  MoveL 1037 to (5.94, 339.15, -10) mm, rotated rx 180 ry 0 rz 0.01 deg; joints [44.933, -47.873, 107.559, -131.107, 69.642, 159.025]
  MoveL 1038 to (6.8, 338.95, -10) mm, rotated rx 180 ry 0 rz 0.01 deg; joints [44.952, -47.906, 107.627, -131.098, 69.673, 159.047]
  MoveL 1039 to (7.07, 338.84, -10) mm, rotated rx 180 ry 0 rz 0.01 deg; joints [44.956, -47.917, 107.651, -131.098, 69.683, 159.056]
  MoveL 1040 to (7.57, 338.46, -9.83) mm, rotated rx -180 ry 0 rz 0.01 deg; joints [44.959, -47.953, 107.708, -131.101, 69.698, 159.072]
  MoveL 1041 to (7.78, 338.05, -9.37) mm, rotated rx -180 ry 0 rz 0.01 deg; joints [44.953, -47.996, 107.749, -131.105, 69.694, 159.072]
  MoveL 1042 to (7.82, 337.88, -8.73) mm, rotated rx 180 ry 0 rz 0.01 deg; joints [44.95, -48.036, 107.764, -131.102, 69.677, 159.053]
  Set speed (500.0 mm/s)
  MoveL 1043 to (7.82, 337.88, 11) mm, rotated rx 180 ry 0 rz 0.01 deg; joints [44.942, -49.073, 107.797, -130.824, 69.015, 158.246]
  Set speed (500.0 mm/s)
  MoveL 1044 to (10.27, 334.35, 11) mm, rotated rx -180 ry 0 rz 0.01 deg; joints [44.912, -49.257, 108.178, -130.911, 69.133, 158.417]
  Set speed (100.0 mm/s)
  MoveL 1045 to (10.27, 334.35, -10) mm, rotated rx 180 ry 0 rz 0.01 deg; joints [44.92, -48.148, 108.142, -131.206, 69.84, 159.277]
  MoveL 1046 to (10.27, 31.58, -10) mm, rotated rx 180 ry 0 rz 0.01 deg; joints [35.104, -55.706, 124.759, -143.156, 73.602, 169.001]
  MoveL 1047 to (8.89, 37.17, -10) mm, rotated rx 180 ry 0 rz 0.01 deg; joints [35.276, -55.549, 124.407, -142.947, 73.483, 168.827]
  MoveL 1048 to (8.76, 37.6, -10) mm, rotated rx 180 ry 0 rz 0.01 deg; joints [35.288, -55.536, 124.378, -142.931, 73.473, 168.813]
  MoveL 1049 to (8.49, 38.29, -10) mm, rotated rx 180 ry 0 rz 0.01 deg; joints [35.306, -55.514, 124.328, -142.908, 73.455, 168.79]
  MoveL 1050 to (8.23, 38.81, -10) mm, rotated rx -180 ry 0 rz 0.01 deg; joints [35.319, -55.495, 124.286, -142.891, 73.439, 168.772]
  MoveL 1051 to (2.04, 48.95, -10) mm, rotated rx 180 ry 0 rz 0.01 deg; joints [35.53, -55.095, 123.399, -142.587, 73.098, 168.4]
  MoveL 1052 to (1.89, 49.17, -10) mm, rotated rx 180 ry 0 rz 0.01 deg; joints [35.534, -55.085, 123.378, -142.581, 73.091, 168.392]
  MoveL 1053 to (1.05, 50.33, -10) mm, rotated rx -180 ry 0 rz 0.01 deg; joints [35.555, -55.035, 123.268, -142.549, 73.047, 168.347]
  MoveL 1054 to (0.43, 50.98, -10) mm, rotated rx 180 ry 0 rz 0.01 deg; joints [35.562, -55.003, 123.196, -142.534, 73.018, 168.32]
  MoveL 1055 to (-7.44, 57.3, -10) mm, rotated rx -180 ry 0 rz 0.01 deg; joints [35.587, -54.626, 122.372, -142.424, 72.668, 168.027]
  MoveL 1056 to (-7.81, 57.56, -10) mm, rotated rx 180 ry 0 rz 0.01 deg; joints [35.587, -54.609, 122.335, -142.421, 72.652, 168.014]
  MoveL 1057 to (-8.49, 57.96, -10) mm, rotated rx -180 ry 0 rz 0.01 deg; joints [35.584, -54.58, 122.271, -142.417, 72.624, 167.993]
  MoveL 1058 to (-9.25, 58.3, -10) mm, rotated rx 180 ry 0 rz 0.01 deg; joints [35.577, -54.549, 122.203, -142.418, 72.594, 167.972]
  MoveL 1059 to (-19.1, 61.27, -10) mm, rotated rx -180 ry 0 rz 0.01 deg; joints [35.43, -54.179, 121.402, -142.484, 72.218, 167.743]
  MoveL 1060 to (-19.95, 61.41, -10) mm, rotated rx -180 ry 0 rz 0.01 deg; joints [35.414, -54.15, 121.339, -142.494, 72.187, 167.726]
  MoveL 1061 to (-21.76, 61.48, -10) mm, rotated rx -180 ry 0 rz 0.01 deg; joints [35.37, -54.091, 121.213, -142.526, 72.123, 167.698]
  MoveL 1062 to (-22.2, 61.47, -10) mm, rotated rx -180 ry 0 rz 0.01 deg; joints [35.358, -54.078, 121.185, -142.534, 72.108, 167.691]
  MoveL 1063 to (-29.46, 60.8, -10) mm, rotated rx -180 ry 0 rz 0.01 deg; joints [35.15, -53.864, 120.726, -142.699, 71.865, 167.604]
  MoveL 1064 to (-29.69, 60.77, -10) mm, rotated rx 180 ry 0 rz 0.01 deg; joints [35.144, -53.857, 120.712, -142.704, 71.857, 167.601]
  MoveL 1065 to (-31.5, 60.48, -10) mm, rotated rx 180 ry 0 rz 0.01 deg; joints [35.087, -53.806, 120.603, -142.75, 71.798, 167.583]
  MoveL 1066 to (-32.21, 60.29, -10) mm, rotated rx 180 ry 0 rz 0.01 deg; joints [35.063, -53.788, 120.565, -142.771, 71.776, 167.578]
  MoveL 1067 to (-34.02, 59.57, -10) mm, rotated rx 180 ry 0 rz 0.01 deg; joints [34.991, -53.745, 120.476, -142.835, 71.722, 167.572]
  MoveL 1068 to (-34.31, 59.44, -10) mm, rotated rx 180 ry 0 rz 0.01 deg; joints [34.979, -53.739, 120.462, -142.846, 71.713, 167.571]
  MoveL 1069 to (-41.06, 55.99, -10) mm, rotated rx -180 ry 0 rz 0.01 deg; joints [34.688, -53.597, 120.166, -143.113, 71.52, 167.57]
  MoveL 1070 to (-41.31, 55.85, -10) mm, rotated rx -180 ry 0 rz 0.01 deg; joints [34.676, -53.592, 120.155, -143.124, 71.513, 167.571]
  MoveL 1071 to (-42.24, 55.27, -10) mm, rotated rx 180 ry 0 rz 0.01 deg; joints [34.632, -53.574, 120.119, -143.165, 71.487, 167.574]
  MoveL 1072 to (-42.6, 55.01, -10) mm, rotated rx 180 ry 0 rz 0.01 deg; joints [34.614, -53.568, 120.106, -143.182, 71.478, 167.576]
  MoveL 1073 to (-43.63, 54.17, -10) mm, rotated rx 180 ry 0 rz 0.01 deg; joints [34.559, -53.553, 120.076, -143.236, 71.452, 167.585]
  MoveL 1074 to (-44.02, 53.79, -10) mm, rotated rx 180 ry 0 rz 0.01 deg; joints [34.535, -53.549, 120.067, -143.259, 71.443, 167.59]
  MoveL 1075 to (-46.92, 50.49, -10) mm, rotated rx -180 ry 0 rz 0.01 deg; joints [34.345, -53.525, 120.023, -143.45, 71.382, 167.641]
  MoveL 1076 to (-46.98, 50.42, -10) mm, rotated rx -180 ry 0 rz 0.01 deg; joints [34.341, -53.524, 120.022, -143.454, 71.381, 167.642]
  MoveL 1077 to (-50.32, 46.42, -10) mm, rotated rx -180 ry 0 rz 0.01 deg; joints [34.116, -53.501, 119.98, -143.682, 71.312, 167.707]
  MoveL 1078 to (-50.64, 45.95, -10) mm, rotated rx -180 ry 0 rz 0.01 deg; joints [34.09, -53.5, 119.979, -143.707, 71.306, 167.716]
  MoveL 1079 to (-68.58, 14.91, -10) mm, rotated rx -180 ry 0 rz 0.01 deg; joints [32.531, -53.548, 120.149, -145.334, 71.045, 168.324]
  MoveL 1080 to (-68.71, 14.67, -10) mm, rotated rx 180 ry 0 rz 0.01 deg; joints [32.519, -53.548, 120.15, -145.347, 71.043, 168.329]
  MoveL 1081 to (-69.4, 13.22, -10) mm, rotated rx 180 ry 0 rz 0.01 deg; joints [32.45, -53.555, 120.167, -145.42, 71.036, 168.36]
  MoveL 1082 to (-69.53, 12.89, -10) mm, rotated rx 180 ry 0 rz 0.01 deg; joints [32.434, -53.557, 120.172, -145.437, 71.035, 168.367]
  MoveL 1083 to (-72.09, 5.64, -10) mm, rotated rx 180 ry 0 rz 0.01 deg; joints [32.107, -53.615, 120.314, -145.79, 71.031, 168.529]
  MoveL 1084 to (-72.16, 5.41, -10) mm, rotated rx -180 ry 0 rz 0.01 deg; joints [32.097, -53.618, 120.319, -145.801, 71.031, 168.535]
  MoveL 1085 to (-72.56, 3.96, -10) mm, rotated rx -180 ry 0 rz 0.01 deg; joints [32.034, -53.633, 120.355, -145.87, 71.034, 168.569]
  MoveL 1086 to (-72.66, 3.43, -10) mm, rotated rx 180 ry 0 rz 0.01 deg; joints [32.012, -53.64, 120.371, -145.894, 71.037, 168.582]
  MoveL 1087 to (-72.82, 1.98, -10) mm, rotated rx -180 ry 0 rz 0.01 deg; joints [31.955, -53.663, 120.423, -145.959, 71.048, 168.619]
  MoveL 1088 to (-72.83, 1.45, -10) mm, rotated rx -180 ry 0 rz 0.01 deg; joints [31.935, -53.672, 120.446, -145.982, 71.054, 168.633]
  MoveL 1089 to (-72.48, -5.8, -10) mm, rotated rx 180 ry 0 rz 0.01 deg; joints [31.673, -53.824, 120.786, -146.288, 71.154, 168.835]
  MoveL 1090 to (-72.47, -5.98, -10) mm, rotated rx 180 ry 0 rz 0.01 deg; joints [31.667, -53.828, 120.795, -146.296, 71.157, 168.84]
  MoveL 1091 to (-72.25, -8.15, -10) mm, rotated rx -180 ry 0 rz 0.01 deg; joints [31.59, -53.876, 120.904, -146.386, 71.191, 168.902]
  MoveL 1092 to (-72.12, -8.81, -10) mm, rotated rx -180 ry 0 rz 0.01 deg; joints [31.569, -53.893, 120.942, -146.412, 71.204, 168.921]
  MoveL 1093 to (-71.7, -10.2, -10) mm, rotated rx 180 ry 0 rz 0.01 deg; joints [31.527, -53.934, 121.032, -146.465, 71.236, 168.965]
  MoveL 1094 to (-71.56, -10.56, -10) mm, rotated rx -180 ry 0 rz 0.01 deg; joints [31.516, -53.945, 121.057, -146.478, 71.245, 168.976]
  MoveL 1095 to (-70.7, -12.52, -10) mm, rotated rx -180 ry 0 rz 0.01 deg; joints [31.462, -54.01, 121.202, -146.549, 71.3, 169.041]
  MoveL 1096 to (-70.68, -12.58, -10) mm, rotated rx 180 ry 0 rz 0.01 deg; joints [31.461, -54.012, 121.207, -146.551, 71.301, 169.043]
  MoveL 1097 to (-68.54, -17.21, -10) mm, rotated rx 180 ry 0 rz 0.01 deg; joints [31.335, -54.17, 121.556, -146.716, 71.435, 169.197]
  MoveL 1098 to (-68.48, -17.34, -10) mm, rotated rx -180 ry 0 rz 0.01 deg; joints [31.332, -54.174, 121.565, -146.72, 71.438, 169.201]
  MoveL 1099 to (-67.74, -18.79, -10) mm, rotated rx 180 ry 0 rz 0.01 deg; joints [31.294, -54.226, 121.68, -146.77, 71.483, 169.25]
  MoveL 1100 to (-67.5, -19.18, -10) mm, rotated rx -180 ry 0 rz 0.01 deg; joints [31.285, -54.241, 121.713, -146.783, 71.496, 169.264]
  MoveL 1101 to (-66.73, -20.29, -10) mm, rotated rx -180 ry 0 rz 0.01 deg; joints [31.26, -54.287, 121.814, -146.819, 71.538, 169.304]
  MoveL 1102 to (-66.27, -20.82, -10) mm, rotated rx 180 ry 0 rz 0.01 deg; joints [31.251, -54.312, 121.869, -146.834, 71.561, 169.325]
  MoveL 1103 to (-59.77, -26.97, -10) mm, rotated rx 180 ry 0 rz 0.01 deg; joints [31.167, -54.638, 122.587, -146.991, 71.871, 169.577]
  MoveL 1104 to (-59.61, -27.11, -10) mm, rotated rx 180 ry 0 rz 0.01 deg; joints [31.165, -54.646, 122.603, -146.994, 71.878, 169.583]
  MoveL 1105 to (-58.52, -28.01, -10) mm, rotated rx 180 ry 0 rz 0.01 deg; joints [31.156, -54.698, 122.718, -147.015, 71.928, 169.622]
  MoveC 1106 to (-58.09, -28.32, -10) mm, rotated rx 180 ry 0 rz 0.01 deg; joints [31.154, -54.718, 122.761, -147.021, 71.948, 169.636] to (-57.61, -28.56, -10) mm, rotated rx 180 ry 0 rz 0.01 deg; joints [31.156, -54.738, 122.805, -147.023, 71.968, 169.649]
  MoveL 1107 to (-50.81, -31.27, -10) mm, rotated rx 180 ry 0 rz 0.01 deg; joints [31.21, -55.008, 123.394, -147.024, 72.247, 169.814]
  MoveL 1108 to (-342.73, -31.27, -10) mm, rotated rx -180 ry 0 rz 0.01 deg; joints [25.542, -44.352, 100.839, -150.359, 60.721, 165.533]
  MoveL 1109 to (-336.29, -28.75, -10) mm, rotated rx 180 ry 0 rz 0.01 deg; joints [25.731, -44.57, 101.289, -150.215, 60.975, 165.561]
  MoveL 1110 to (-335.78, -28.5, -10) mm, rotated rx 180 ry 0 rz 0.01 deg; joints [25.748, -44.586, 101.323, -150.201, 60.994, 165.562]
  MoveL 1111 to (-335.05, -28.07, -10) mm, rotated rx -180 ry 0 rz 0.01 deg; joints [25.774, -44.608, 101.367, -150.178, 61.021, 165.56]
  MoveL 1112 to (-334.49, -27.65, -10) mm, rotated rx -180 ry 0 rz 0.01 deg; joints [25.798, -44.623, 101.398, -150.157, 61.041, 165.556]
  MoveL 1113 to (-332.31, -25.62, -10) mm, rotated rx 180 ry 0 rz 0.01 deg; joints [25.902, -44.674, 101.5, -150.057, 61.114, 165.529]
  MoveL 1114 to (-332.27, -25.59, -10) mm, rotated rx -180 ry 0 rz 0.01 deg; joints [25.904, -44.675, 101.502, -150.055, 61.115, 165.529]
  MoveL 1115 to (-326.92, -20.45, -10) mm, rotated rx 180 ry 0 rz 0.01 deg; joints [26.166, -44.796, 101.745, -149.801, 61.293, 165.457]
  MoveL 1116 to (-326.37, -19.77, -10) mm, rotated rx 180 ry 0 rz 0.01 deg; joints [26.198, -44.805, 101.764, -149.768, 61.309, 165.445]
  MoveL 1117 to (-325.69, -18.65, -10) mm, rotated rx 180 ry 0 rz 0.01 deg; joints [26.247, -44.812, 101.775, -149.716, 61.327, 165.421]
  MoveL 1118 to (-325.51, -18.31, -10) mm, rotated rx 180 ry 0 rz 0.01 deg; joints [26.262, -44.813, 101.776, -149.7, 61.331, 165.414]
  MoveL 1119 to (-322.24, -11.28, -10) mm, rotated rx 180 ry 0 rz 0.01 deg; joints [26.553, -44.81, 101.758, -149.376, 61.398, 165.248]
  MoveL 1120 to (-322.12, -11.01, -10) mm, rotated rx -180 ry 0 rz 0.01 deg; joints [26.565, -44.81, 101.756, -149.363, 61.4, 165.241]
  MoveL 1121 to (-321.52, -9.33, -10) mm, rotated rx -180 ry 0 rz 0.01 deg; joints [26.631, -44.802, 101.736, -149.287, 61.408, 165.199]
  MoveL 1122 to (-321.34, -8.57, -10) mm, rotated rx -180 ry 0 rz 0.01 deg; joints [26.66, -44.794, 101.719, -149.253, 61.408, 165.178]
  MoveL 1123 to (-321.05, -6.03, -10) mm, rotated rx -180 ry 0 rz 0.01 deg; joints [26.75, -44.757, 101.635, -149.142, 61.394, 165.103]
  MoveL 1124 to (-321.03, -5.8, -10) mm, rotated rx -180 ry 0 rz 0.01 deg; joints [26.758, -44.753, 101.627, -149.132, 61.392, 165.096]
  MoveL 1125 to (-320.68, 1.45, -10) mm, rotated rx 180 ry 0 rz 0.01 deg; joints [27.007, -44.624, 101.345, -148.816, 61.331, 164.873]
  MoveL 1126 to (-320.69, 1.86, -10) mm, rotated rx -180 ry 0 rz 0.01 deg; joints [27.021, -44.616, 101.327, -148.799, 61.327, 164.86]
  MoveL 1127 to (-320.74, 2.59, -10) mm, rotated rx -180 ry 0 rz 0.01 deg; joints [27.044, -44.599, 101.291, -148.768, 61.317, 164.836]
  MoveL 1128 to (-320.78, 2.94, -10) mm, rotated rx -180 ry 0 rz 0.01 deg; joints [27.055, -44.59, 101.272, -148.753, 61.311, 164.824]
  MoveL 1129 to (-321.05, 4.39, -10) mm, rotated rx 180 ry 0 rz 0.01 deg; joints [27.099, -44.551, 101.187, -148.692, 61.285, 164.773]
  MoveL 1130 to (-321.17, 4.88, -10) mm, rotated rx -180 ry 0 rz 0.01 deg; joints [27.113, -44.536, 101.155, -148.671, 61.274, 164.756]
  MoveL 1131 to (-321.92, 7.06, -10) mm, rotated rx 180 ry 0 rz 0.01 deg; joints [27.173, -44.462, 100.997, -148.582, 61.219, 164.674]
  MoveL 1132 to (-321.94, 7.11, -10) mm, rotated rx 180 ry 0 rz 0.01 deg; joints [27.175, -44.46, 100.993, -148.58, 61.218, 164.672]
  MoveL 1133 to (-324.29, 13.64, -10) mm, rotated rx 180 ry 0 rz 0.01 deg; joints [27.351, -44.233, 100.506, -148.312, 61.048, 164.422]
  MoveL 1134 to (-324.54, 14.18, -10) mm, rotated rx -180 ry 0 rz 0.01 deg; joints [27.365, -44.212, 100.461, -148.29, 61.032, 164.4]
  MoveL 1135 to (-342.52, 45.38, -10) mm, rotated rx -180 ry 0 rz 0.01 deg; joints [28.076, -42.818, 97.505, -147.038, 59.927, 163.048]
  MoveL 1136 to (-342.66, 45.6, -10) mm, rotated rx 180 ry 0 rz 0.01 deg; joints [28.081, -42.808, 97.483, -147.029, 59.919, 163.038]
  MoveL 1137 to (-343.43, 46.73, -10) mm, rotated rx 180 ry 0 rz 0.01 deg; joints [28.104, -42.751, 97.363, -146.983, 59.873, 162.985]
  MoveL 1138 to (-343.65, 47.02, -10) mm, rotated rx -180 ry 0 rz 0.01 deg; joints [28.11, -42.736, 97.33, -146.972, 59.861, 162.971]
  MoveL 1139 to (-348.97, 53.24, -10) mm, rotated rx 180 ry 0 rz 0.01 deg; joints [28.218, -42.378, 96.576, -146.726, 59.563, 162.659]
  MoveL 1140 to (-349.18, 53.47, -10) mm, rotated rx 180 ry 0 rz 0.01 deg; joints [28.222, -42.364, 96.547, -146.718, 59.552, 162.647]
  MoveL 1141 to (-350.19, 54.44, -10) mm, rotated rx 180 ry 0 rz 0.01 deg; joints [28.236, -42.3, 96.413, -146.68, 59.498, 162.595]
  MoveL 1142 to (-350.57, 54.76, -10) mm, rotated rx -180 ry 0 rz 0.01 deg; joints [28.239, -42.277, 96.365, -146.667, 59.477, 162.576]
  MoveL 1143 to (-351.55, 55.47, -10) mm, rotated rx 180 ry 0 rz 0.01 deg; joints [28.245, -42.22, 96.245, -146.641, 59.427, 162.533]
  MoveL 1144 to (-351.98, 55.73, -10) mm, rotated rx -180 ry 0 rz 0.01 deg; joints [28.246, -42.197, 96.196, -146.631, 59.406, 162.516]
  MoveL 1145 to (-359.19, 59.43, -10) mm, rotated rx -180 ry 0 rz 0.01 deg; joints [28.241, -41.809, 95.384, -146.498, 59.051, 162.248]
  MoveL 1146 to (-359.41, 59.54, -10) mm, rotated rx -180 ry 0 rz 0.01 deg; joints [28.24, -41.797, 95.36, -146.495, 59.04, 162.24]
  MoveL 1147 to (-360.86, 60.15, -10) mm, rotated rx 180 ry 0 rz 0.01 deg; joints [28.235, -41.721, 95.202, -146.473, 58.97, 162.19]
  MoveL 1148 to (-361.5, 60.35, -10) mm, rotated rx -180 ry 0 rz 0.01 deg; joints [28.23, -41.69, 95.136, -146.467, 58.94, 162.17]
  MoveL 1149 to (-362.95, 60.65, -10) mm, rotated rx 180 ry 0 rz 0.01 deg; joints [28.215, -41.621, 94.993, -146.458, 58.873, 162.131]
  MoveL 1150 to (-363.32, 60.71, -10) mm, rotated rx 180 ry 0 rz 0.01 deg; joints [28.211, -41.604, 94.957, -146.457, 58.856, 162.122]
  MoveL 1151 to (-371.3, 61.47, -10) mm, rotated rx -180 ry 0 rz 0.01 deg; joints [28.099, -41.243, 94.209, -146.45, 58.495, 161.936]
  MoveL 1152 to (-371.75, 61.48, -10) mm, rotated rx -180 ry 0 rz 0.01 deg; joints [28.092, -41.224, 94.168, -146.451, 58.476, 161.927]
  MoveL 1153 to (-373.56, 61.41, -10) mm, rotated rx 180 ry 0 rz 0.01 deg; joints [28.059, -41.147, 94.009, -146.459, 58.396, 161.892]
  MoveL 1154 to (-374.4, 61.27, -10) mm, rotated rx -180 ry 0 rz 0.01 deg; joints [28.041, -41.114, 93.94, -146.467, 58.36, 161.88]
  MoveL 1155 to (-383.58, 58.54, -10) mm, rotated rx -180 ry 0 rz 0.01 deg; joints [27.801, -40.774, 93.242, -146.61, 57.981, 161.79]
  MoveL 1156 to (-383.9, 58.43, -10) mm, rotated rx 180 ry 0 rz 0.01 deg; joints [27.793, -40.762, 93.218, -146.616, 57.968, 161.788]
  MoveL 1157 to (-384.9, 58.02, -10) mm, rotated rx 180 ry 0 rz 0.01 deg; joints [27.763, -40.728, 93.147, -146.636, 57.927, 161.782]
  MoveL 1158 to (-385.72, 57.54, -10) mm, rotated rx 180 ry 0 rz 0.01 deg; joints [27.734, -40.702, 93.095, -146.659, 57.896, 161.782]
  MoveL 1159 to (-393.23, 51.6, -10) mm, rotated rx -180 ry 0 rz 0.01 deg; joints [27.424, -40.503, 92.693, -146.935, 57.622, 161.838]
  MoveL 1160 to (-393.47, 51.39, -10) mm, rotated rx 180 ry 0 rz 0.01 deg; joints [27.413, -40.497, 92.681, -146.944, 57.613, 161.841]
  MoveL 1161 to (-394.4, 50.5, -10) mm, rotated rx -180 ry 0 rz 0.01 deg; joints [27.37, -40.475, 92.637, -146.985, 57.581, 161.853]
  MoveL 1162 to (-394.94, 49.84, -10) mm, rotated rx 180 ry 0 rz 0.01 deg; joints [27.34, -40.466, 92.62, -147.015, 57.563, 161.866]
  MoveL 1163 to (-401.25, 39.67, -10) mm, rotated rx 180 ry 0 rz 0.01 deg; joints [26.917, -40.408, 92.518, -147.474, 57.386, 162.097]
  MoveL 1164 to (-401.38, 39.45, -10) mm, rotated rx 180 ry 0 rz 0.01 deg; joints [26.908, -40.408, 92.517, -147.483, 57.382, 162.102]
  MoveL 1165 to (-401.99, 38.27, -10) mm, rotated rx -180 ry 0 rz 0.01 deg; joints [26.861, -40.406, 92.515, -147.536, 57.367, 162.131]
  MoveL 1166 to (-402.27, 37.54, -10) mm, rotated rx 180 ry 0 rz 0.01 deg; joints [26.833, -40.409, 92.523, -147.569, 57.362, 162.151]
  MoveL 1167 to (-403.78, 31.65, -10) mm, rotated rx 180 ry 0 rz 0.01 deg; joints [26.622, -40.469, 92.658, -147.831, 57.356, 162.328]
  MoveL 1168 to (-403.79, 333.8, -10) mm, rotated rx 180 ry 0 rz 0.01 deg; joints [35.399, -32.082, 74.938, -134.135, 53.84, 149.634]
  MoveL 1169 to (-403.73, 334.87, -10) mm, rotated rx -180 ry 0 rz 0.01 deg; joints [35.429, -32.047, 74.865, -134.084, 53.829, 149.582]
  MoveL 1170 to (-403.53, 335.74, -10) mm, rotated rx -180 ry 0 rz 0.01 deg; joints [35.455, -32.027, 74.822, -134.044, 53.827, 149.545]
  MoveL 1171 to (-403.42, 336, -10) mm, rotated rx -180 ry 0 rz 0.01 deg; joints [35.464, -32.023, 74.814, -134.032, 53.829, 149.535]
  MoveL 1172 to (-403.03, 336.5, -9.83) mm, rotated rx -180 ry 0 rz 0.01 deg; joints [35.485, -32.032, 74.818, -134.008, 53.836, 149.518]
  MoveL 1173 to (-402.62, 336.71, -9.37) mm, rotated rx -180 ry 0 rz 0.01 deg; joints [35.498, -32.064, 74.846, -133.992, 53.84, 149.506]
  MoveL 1174 to (-402.46, 336.75, -8.73) mm, rotated rx -180 ry 0 rz 0.01 deg; joints [35.502, -32.098, 74.862, -133.979, 53.83, 149.488]
  Set speed (500.0 mm/s)
  MoveL 1175 to (-402.46, 336.75, 11) mm, rotated rx 180 ry 0 rz 0.01 deg; joints [35.493, -32.912, 74.899, -133.574, 53.288, 148.796]
  Set speed (500.0 mm/s)
  MoveL 1176 to (-182.2, 109.36, 11) mm, rotated rx 180 ry 0 rz 0.01 deg; joints [33.246, -48.741, 107.487, -142.719, 64.876, 163.062]
  Set speed (500.0 mm/s)
  MoveL 1177 to (-182.2, 109.36, 1.77) mm, rotated rx 180 ry 0 rz 0.01 deg; joints [33.251, -48.259, 107.475, -142.846, 65.252, 163.373]
  Set speed (100.0 mm/s)
  MoveL 1178 to (-182.04, 109.34, 1.15) mm, rotated rx 180 ry 0 rz 0.01 deg; joints [33.254, -48.233, 107.487, -142.853, 65.284, 163.397]
  MoveL 1179 to (-181.59, 109.31, 0.68) mm, rotated rx -180 ry 0 rz 0.01 deg; joints [33.263, -48.226, 107.521, -142.855, 65.32, 163.421]
  MoveL 1180 to (-180.98, 109.33, 0.5) mm, rotated rx -180 ry 0 rz 0.01 deg; joints [33.277, -48.238, 107.567, -142.85, 65.35, 163.437]
  MoveL 1181 to (-175.74, 113.35, 0.26) mm, rotated rx -180 ry 0 rz 0.01 deg; joints [33.523, -48.323, 107.762, -142.624, 65.514, 163.401]
  MoveL 1182 to (-177.33, 119.76, 0.01) mm, rotated rx 180 ry 0 rz 0.01 deg; joints [33.698, -48.103, 107.32, -142.379, 65.392, 163.174]
  MoveL 1183 to (-183.84, 120.88, -0.23) mm, rotated rx -180 ry 0 rz 0.01 deg; joints [33.593, -47.827, 106.771, -142.412, 65.143, 163.038]
  MoveL 1184 to (-187.47, 115.36, -0.48) mm, rotated rx -180 ry 0 rz 0.01 deg; joints [33.336, -47.81, 106.772, -142.686, 65.077, 163.166]
  MoveL 1185 to (-183.86, 109.82, -0.72) mm, rotated rx -180 ry 0 rz 0.01 deg; joints [33.232, -48.057, 107.321, -142.879, 65.285, 163.414]
  MoveL 1186 to (-177.35, 110.91, -0.96) mm, rotated rx -180 ry 0 rz 0.01 deg; joints [33.408, -48.257, 107.76, -142.761, 65.53, 163.494]
  MoveL 1187 to (-175.73, 117.31, -1.21) mm, rotated rx -180 ry 0 rz 0.01 deg; joints [33.653, -48.154, 107.562, -142.479, 65.529, 163.322]
  MoveL 1188 to (-180.95, 121.36, -1.45) mm, rotated rx -180 ry 0 rz 0.01 deg; joints [33.672, -47.857, 106.963, -142.375, 65.296, 163.111]
  MoveL 1189 to (-186.75, 118.2, -1.7) mm, rotated rx -180 ry 0 rz 0.01 deg; joints [33.444, -47.706, 106.682, -142.576, 65.121, 163.126]
  MoveL 1190 to (-186.18, 111.62, -1.94) mm, rotated rx -180 ry 0 rz 0.01 deg; joints [33.242, -47.867, 107.053, -142.847, 65.226, 163.358]
  MoveL 1191 to (-179.92, 109.5, -2.18) mm, rotated rx 180 ry 0 rz 0.01 deg; joints [33.307, -48.131, 107.633, -142.866, 65.497, 163.538]
  MoveL 1192 to (-175.48, 114.39, -2.43) mm, rotated rx -180 ry 0 rz 0.01 deg; joints [33.564, -48.167, 107.724, -142.613, 65.621, 163.462]
  MoveL 1193 to (-178.17, 120.42, -2.67) mm, rotated rx 180 ry 0 rz 0.01 deg; joints [33.702, -47.916, 107.218, -142.398, 65.461, 163.229]
  MoveL 1194 to (-184.77, 120.37, -2.92) mm, rotated rx 180 ry 0 rz 0.01 deg; joints [33.558, -47.664, 106.72, -142.48, 65.221, 163.129]
  MoveL 1195 to (-187.37, 114.3, -3.16) mm, rotated rx 180 ry 0 rz 0.01 deg; joints [33.304, -47.698, 106.826, -142.766, 65.2, 163.292]
  MoveL 1196 to (-182.85, 109.48, -3.4) mm, rotated rx -180 ry 0 rz 0.01 deg; joints [33.244, -47.961, 107.409, -142.918, 65.436, 163.531]
  MoveL 1197 to (-176.63, 111.69, -3.65) mm, rotated rx -180 ry 0 rz 0.01 deg; joints [33.451, -48.123, 107.769, -142.756, 65.657, 163.57]
  MoveL 1198 to (-176.16, 118.28, -3.89) mm, rotated rx 180 ry 0 rz 0.01 deg; joints [33.677, -47.975, 107.475, -142.479, 65.61, 163.373]
  MoveL 1199 to (-182.01, 121.35, -4.14) mm, rotated rx 180 ry 0 rz 0.01 deg; joints [33.65, -47.678, 106.878, -142.424, 65.363, 163.184]
  MoveL 1200 to (-187.17, 117.22, -4.38) mm, rotated rx -180 ry 0 rz 0.01 deg; joints [33.405, -47.574, 106.693, -142.658, 65.224, 163.24]
  MoveL 1201 to (-185.45, 110.84, -4.63) mm, rotated rx 180 ry 0 rz 0.01 deg; joints [33.234, -47.771, 107.142, -142.907, 65.371, 163.484]
  MoveL 1202 to (-178.92, 109.86, -4.87) mm, rotated rx -180 ry 0 rz 0.01 deg; joints [33.342, -48.018, 107.685, -142.875, 65.64, 163.632]
  MoveL 1203 to (-175.4, 115.45, -5.11) mm, rotated rx 180 ry 0 rz 0.01 deg; joints [33.602, -48.003, 107.671, -142.604, 65.72, 163.518]
  MoveL 1204 to (-179.11, 120.91, -5.36) mm, rotated rx -180 ry 0 rz 0.01 deg; joints [33.699, -47.73, 107.116, -142.424, 65.527, 163.287]
  MoveL 1205 to (-185.61, 119.7, -5.6) mm, rotated rx 180 ry 0 rz 0.01 deg; joints [33.52, -47.509, 106.685, -142.553, 65.304, 163.226]
  MoveL 1206 to (-187.1, 113.27, -5.85) mm, rotated rx -180 ry 0 rz 0.01 deg; joints [33.278, -47.591, 106.893, -142.841, 65.33, 163.419]
  MoveL 1207 to (-181.8, 109.32, -6.09) mm, rotated rx -180 ry 0 rz 0.01 deg; joints [33.263, -47.861, 107.491, -142.948, 65.586, 163.643]
  MoveL 1208 to (-176.06, 112.6, -6.33) mm, rotated rx -180 ry 0 rz 0.01 deg; joints [33.494, -47.981, 107.761, -142.747, 65.777, 163.64]
  MoveL 1209 to (-176.76, 119.16, -6.58) mm, rotated rx -180 ry 0 rz 0.01 deg; joints [33.694, -47.791, 107.379, -142.486, 65.685, 163.424]
  MoveL 1210 to (-183.06, 121.15, -6.82) mm, rotated rx 180 ry 0 rz 0.01 deg; joints [33.623, -47.504, 106.802, -142.48, 65.433, 163.262]
  MoveL 1211 to (-187.41, 116.18, -7.07) mm, rotated rx 180 ry 0 rz 0.01 deg; joints [33.367, -47.448, 106.721, -142.74, 65.333, 163.359]
  MoveL 1212 to (-184.59, 110.21, -7.31) mm, rotated rx -180 ry 0 rz 0.01 deg; joints [33.233, -47.675, 107.232, -142.959, 65.519, 163.608]
  MoveL 1213 to (-177.99, 110.39, -7.55) mm, rotated rx -180 ry 0 rz 0.01 deg; joints [33.381, -47.897, 107.723, -142.877, 65.778, 163.72]
  MoveL 1214 to (-175.52, 116.51, -7.8) mm, rotated rx 180 ry 0 rz 0.01 deg; joints [33.635, -47.833, 107.603, -142.597, 65.812, 163.572]
  MoveL 1215 to (-180.13, 121.24, -8.04) mm, rotated rx -180 ry 0 rz 0.01 deg; joints [33.689, -47.544, 107.017, -142.459, 65.592, 163.349]
  MoveL 1216 to (-186.31, 118.9, -8.29) mm, rotated rx 180 ry 0 rz 0.01 deg; joints [33.48, -47.362, 106.665, -142.631, 65.393, 163.329]
  MoveL 1217 to (-186.64, 112.3, -8.53) mm, rotated rx 180 ry 0 rz 0.01 deg; joints [33.258, -47.489, 106.969, -142.912, 65.466, 163.546]
  MoveL 1218 to (-180.73, 109.35, -8.77) mm, rotated rx 180 ry 0 rz 0.01 deg; joints [33.288, -47.758, 107.564, -142.969, 65.735, 163.748]
  MoveL 1219 to (-175.66, 113.59, -9.02) mm, rotated rx -180 ry 0 rz 0.01 deg; joints [33.537, -47.831, 107.735, -142.736, 65.889, 163.704]
  MoveL 1220 to (-177.51, 119.93, -9.26) mm, rotated rx 180 ry 0 rz 0.01 deg; joints [33.704, -47.605, 107.278, -142.498, 65.755, 163.476]
  MoveL 1221 to (-184.06, 120.78, -9.51) mm, rotated rx -180 ry 0 rz 0.01 deg; joints [33.59, -47.336, 106.738, -142.543, 65.506, 163.347]
  MoveL 1222 to (-187.46, 115.12, -9.75) mm, rotated rx -180 ry 0 rz 0.01 deg; joints [33.333, -47.33, 106.763, -142.82, 65.451, 163.481]
  MoveL 1223 to (-183.64, 109.73, -9.99) mm, rotated rx 180 ry 0 rz 0.01 deg; joints [33.239, -47.579, 107.322, -143.003, 65.669, 163.728]
  MoveL 1224 to (-177.17, 111.07, -10.24) mm, rotated rx 180 ry 0 rz 0.01 deg; joints [33.423, -47.769, 107.743, -142.874, 65.91, 163.8]
  MoveL 1225 to (-175.81, 117.54, -10.48) mm, rotated rx 180 ry 0 rz 0.01 deg; joints [33.664, -47.657, 107.522, -142.593, 65.896, 163.623]
  MoveL 1226 to (-181.19, 121.37, -10.73) mm, rotated rx -180 ry 0 rz 0.01 deg; joints [33.672, -47.362, 106.923, -142.501, 65.657, 163.416]
  MoveL 1227 to (-186.86, 117.98, -10.97) mm, rotated rx 180 ry 0 rz 0.01 deg; joints [33.44, -47.222, 106.662, -142.711, 65.489, 163.438]
  MoveL 1228 to (-186.03, 111.43, -11.21) mm, rotated rx -180 ry 0 rz 0.01 deg; joints [33.244, -47.39, 107.052, -142.976, 65.607, 163.673]
  MoveL 1229 to (-179.69, 109.57, -11.46) mm, rotated rx -180 ry 0 rz 0.01 deg; joints [33.32, -47.648, 107.625, -142.983, 65.88, 163.847]
  MoveL 1230 to (-175.44, 114.63, -11.7) mm, rotated rx 180 ry 0 rz 0.01 deg; joints [33.577, -47.672, 107.693, -142.725, 65.993, 163.763]
  MoveL 1231 to (-178.38, 120.55, -11.95) mm, rotated rx -180 ry 0 rz 0.01 deg; joints [33.707, -47.418, 107.174, -142.518, 65.822, 163.531]
  MoveL 1232 to (-184.97, 120.23, -12.19) mm, rotated rx 180 ry 0 rz 0.01 deg; joints [33.554, -47.174, 106.689, -142.612, 65.584, 163.437]
  MoveL 1233 to (-187.33, 114.06, -12.43) mm, rotated rx -180 ry 0 rz 0.01 deg; joints [33.303, -47.218, 106.819, -142.898, 65.575, 163.606]
  MoveL 1234 to (-182.62, 109.43, -12.68) mm, rotated rx -180 ry 0 rz 0.01 deg; joints [33.253, -47.481, 107.407, -143.039, 65.819, 163.843]
  MoveL 1235 to (-176.49, 111.89, -12.92) mm, rotated rx -180 ry 0 rz 0.01 deg; joints [33.466, -47.633, 107.747, -142.867, 66.034, 163.874]
  MoveL 1236 to (-176.29, 118.49, -13.17) mm, rotated rx 180 ry 0 rz 0.01 deg; joints [33.686, -47.476, 107.431, -142.594, 65.975, 163.673]
  MoveL 1237 to (-182.26, 121.32, -13.41) mm, rotated rx -180 ry 0 rz 0.01 deg; joints [33.649, -47.183, 106.837, -142.551, 65.724, 163.488]
  MoveL 1238 to (-187.24, 116.99, -13.65) mm, rotated rx 180 ry 0 rz 0.01 deg; joints [33.401, -47.09, 106.676, -142.791, 65.593, 163.552]
  MoveL 1239 to (-185.26, 110.68, -13.9) mm, rotated rx -180 ry 0 rz 0.01 deg; joints [33.237, -47.293, 107.14, -143.033, 65.752, 163.798]
  MoveL 1240 to (-178.7, 109.97, -14.14) mm, rotated rx -180 ry 0 rz 0.01 deg; joints [33.355, -47.532, 107.672, -142.989, 66.021, 163.939]
  MoveL 1241 to (-175.41, 115.7, -14.39) mm, rotated rx 180 ry 0 rz 0.01 deg; joints [33.615, -47.506, 107.634, -142.715, 66.089, 163.818]
  MoveL 1242 to (-179.34, 121, -14.63) mm, rotated rx 180 ry 0 rz 0.01 deg; joints [33.702, -47.231, 107.07, -142.546, 65.887, 163.588]
  MoveL 1243 to (-185.78, 119.53, -14.87) mm, rotated rx -180 ry 0 rz 0.01 deg; joints [33.515, -47.02, 106.655, -142.685, 65.668, 163.535]
  MoveL 1244 to (-187.01, 113.04, -15.12) mm, rotated rx 180 ry 0 rz 0.01 deg; joints [33.278, -47.112, 106.886, -142.972, 65.706, 163.732]
  MoveL 1245 to (-181.56, 109.31, -15.36) mm, rotated rx 180 ry 0 rz 0.01 deg; joints [33.273, -47.38, 107.485, -143.066, 65.969, 163.952]
  MoveL 1246 to (-175.96, 112.82, -15.61) mm, rotated rx -180 ry 0 rz 0.01 deg; joints [33.509, -47.488, 107.733, -142.857, 66.151, 163.942]
  MoveL 1247 to (-176.92, 119.35, -15.85) mm, rotated rx -180 ry 0 rz 0.01 deg; joints [33.702, -47.291, 107.332, -142.601, 66.047, 163.723]
  MoveL 1248 to (-183.29, 121.08, -16.1) mm, rotated rx 180 ry 0 rz 0.01 deg; joints [33.62, -47.01, 106.762, -142.608, 65.793, 163.567]
  MoveL 1249 to (-187.44, 115.94, -16.34) mm, rotated rx 180 ry 0 rz 0.01 deg; joints [33.364, -46.965, 106.705, -142.872, 65.704, 163.671]
  MoveL 1250 to (-184.38, 110.08, -16.58) mm, rotated rx 180 ry 0 rz 0.01 deg; joints [33.238, -47.196, 107.228, -143.083, 65.9, 163.919]
  MoveL 1251 to (-177.79, 110.53, -16.83) mm, rotated rx 180 ry 0 rz 0.01 deg; joints [33.395, -47.409, 107.704, -142.989, 66.157, 164.024]
  MoveL 1252 to (-175.57, 116.75, -17.07) mm, rotated rx -180 ry 0 rz 0.01 deg; joints [33.647, -47.334, 107.561, -142.708, 66.178, 163.87]
  MoveL 1253 to (-180.37, 121.28, -17.32) mm, rotated rx 180 ry 0 rz 0.01 deg; joints [33.691, -47.045, 106.97, -142.581, 65.951, 163.65]
  MoveL 1254 to (-186.45, 118.7, -17.56) mm, rotated rx -180 ry 0 rz 0.01 deg; joints [33.476, -46.874, 106.638, -142.762, 65.758, 163.638]
  MoveL 1255 to (-186.52, 112.09, -17.8) mm, rotated rx -180 ry 0 rz 0.01 deg; joints [33.259, -47.009, 106.962, -143.04, 65.843, 163.858]
  MoveL 1256 to (-180.49, 109.39, -18.05) mm, rotated rx 180 ry 0 rz 0.01 deg; joints [33.3, -47.273, 107.553, -143.084, 66.117, 164.055]
  MoveL 1257 to (-175.6, 113.82, -18.29) mm, rotated rx -180 ry 0 rz 0.01 deg; joints [33.551, -47.335, 107.701, -142.845, 66.261, 164.004]
  MoveL 1258 to (-177.7, 120.08, -18.54) mm, rotated rx 180 ry 0 rz 0.01 deg; joints [33.71, -47.104, 107.228, -142.615, 66.116, 163.774]
  MoveL 1259 to (-184.28, 120.67, -18.78) mm, rotated rx 180 ry 0 rz 0.01 deg; joints [33.587, -46.842, 106.7, -142.671, 65.866, 163.651]
  MoveL 1260 to (-187.45, 114.87, -19.02) mm, rotated rx 180 ry 0 rz 0.01 deg; joints [33.33, -46.848, 106.749, -142.951, 65.823, 163.792]
  MoveL 1261 to (-183.41, 109.65, -19.27) mm, rotated rx -180 ry 0 rz 0.01 deg; joints [33.246, -47.098, 107.315, -143.124, 66.05, 164.037]
  MoveL 1262 to (-177, 111.25, -19.51) mm, rotated rx 180 ry 0 rz 0.01 deg; joints [33.437, -47.278, 107.719, -142.984, 66.287, 164.102]
  MoveL 1263 to (-175.91, 117.76, -19.76) mm, rotated rx 180 ry 0 rz 0.01 deg; joints [33.674, -47.156, 107.476, -142.704, 66.26, 163.92]
  MoveL 1264 to (-181.43, 121.38, -20) mm, rotated rx -180 ry 0 rz 0.01 deg; joints [33.672, -46.863, 106.875, -142.624, 66.015, 163.717]
  MoveL 1265 to (-213.98, 121.38, -20) mm, rotated rx 180 ry 0 rz 0.01 deg; joints [32.98, -45.681, 104.376, -142.983, 64.753, 163.15]
  MoveC 1266 to (-215.9, 120.27, -20) mm, rotated rx 180 ry 0 rz 0.01 deg; joints [32.904, -45.636, 104.282, -143.049, 64.69, 163.153] to (-215.9, 118.04, -20) mm, rotated rx -180 ry 0 rz 0.01 deg; joints [32.833, -45.687, 104.394, -143.142, 64.717, 163.226]
  MoveL 1267 to (-214.81, 116.14, -20) mm, rotated rx 180 ry 0 rz 0.01 deg; joints [32.794, -45.771, 104.575, -143.21, 64.782, 163.308]
  MoveC 1268 to (-213.77, 115.1, -20) mm, rotated rx 180 ry 0 rz 0.01 deg; joints [32.782, -45.833, 104.708, -143.242, 64.835, 163.36] to (-212.35, 114.72, -20) mm, rotated rx -180 ry 0 rz 0.01 deg; joints [32.799, -45.894, 104.838, -143.243, 64.895, 163.397]
  MoveL 1269 to (-181.15, 114.72, -20) mm, rotated rx 180 ry 0 rz 0.01 deg; joints [33.461, -47.025, 107.231, -142.896, 66.106, 163.936]
  MoveC 1270 to (-179.73, 115.1, -20) mm, rotated rx 180 ry 0 rz 0.01 deg; joints [33.505, -47.067, 107.319, -142.863, 66.156, 163.948] to (-178.69, 116.14, -20) mm, rotated rx 180 ry 0 rz 0.01 deg; joints [33.561, -47.081, 107.346, -142.808, 66.183, 163.932]
  MoveL 1271 to (-177.6, 118.04, -20) mm, rotated rx 180 ry 0 rz 0.01 deg; joints [33.647, -47.077, 107.334, -142.716, 66.202, 163.89]
  MoveC 1272 to (-177.59, 120.26, -20) mm, rotated rx 180 ry 0 rz 0.01 deg; joints [33.719, -47.026, 107.222, -142.624, 66.176, 163.818] to (-179.52, 121.38, -20) mm, rotated rx 180 ry 0 rz 0.01 deg; joints [33.714, -46.932, 107.02, -142.601, 66.088, 163.749]
  MoveL 1273 to (-181.43, 121.38, -20) mm, rotated rx -180 ry 0 rz 0.01 deg; joints [33.672, -46.863, 106.875, -142.624, 66.015, 163.717]
  MoveC 1274 to (-184.81, 122.4, -20) mm, rotated rx 180 ry 0 rz 0.01 deg; joints [33.632, -46.719, 106.568, -142.621, 65.873, 163.626] to (-187.05, 125.12, -20) mm, rotated rx 180 ry 0 rz 0.01 deg; joints [33.672, -46.576, 106.26, -142.535, 65.755, 163.498]
  MoveC 1275 to (-189.29, 127.84, -20) mm, rotated rx 180 ry 0 rz 0.01 deg; joints [33.712, -46.432, 105.951, -142.448, 65.636, 163.37] to (-192.66, 128.86, -20) mm, rotated rx 180 ry 0 rz 0.01 deg; joints [33.672, -46.286, 105.641, -142.444, 65.494, 163.278]
  MoveL 1276 to (-214.9, 128.86, -20) mm, rotated rx 180 ry 0 rz 0.01 deg; joints [33.201, -45.473, 103.925, -142.682, 64.628, 162.886]
  MoveC 1277 to (-218.57, 128.97, -20) mm, rotated rx -180 ry 0 rz 0.01 deg; joints [33.128, -45.335, 103.633, -142.715, 64.483, 162.816] to (-222.23, 129.28, -20) mm, rotated rx -180 ry 0 rz 0.01 deg; joints [33.062, -45.191, 103.33, -142.738, 64.334, 162.74]
  MoveC 1278 to (-225.89, 129.69, -20) mm, rotated rx 180 ry 0 rz 0.01 deg; joints [32.999, -45.046, 103.022, -142.756, 64.185, 162.66] to (-229.54, 130.08, -20) mm, rotated rx 180 ry 0 rz 0.01 deg; joints [32.936, -44.9, 102.713, -142.775, 64.036, 162.581]
  MoveC 1279 to (-231.34, 129.16, -20) mm, rotated rx -180 ry 0 rz 0.01 deg; joints [32.87, -44.854, 102.618, -142.83, 63.975, 162.579] to (-231.23, 127.15, -20) mm, rotated rx -180 ry 0 rz 0.01 deg; joints [32.808, -44.905, 102.73, -142.913, 64.003, 162.649]
  MoveC 1280 to (-228.5, 123.23, -20) mm, rotated rx 180 ry 0 rz 0.01 deg; joints [32.739, -45.098, 103.144, -143.051, 64.158, 162.829] to (-225.92, 119.22, -20) mm, rotated rx 180 ry 0 rz 0.01 deg; joints [32.663, -45.288, 103.55, -143.193, 64.308, 163.009]
  MoveC 1281 to (-223.44, 115.14, -20) mm, rotated rx 180 ry 0 rz 0.01 deg; joints [32.583, -45.474, 103.95, -143.339, 64.454, 163.188] to (-221.03, 111.02, -20) mm, rotated rx 180 ry 0 rz 0.01 deg; joints [32.5, -45.657, 104.345, -143.486, 64.597, 163.366]
  MoveC 1282 to (-217.92, 107.91, -20) mm, rotated rx 180 ry 0 rz 0.01 deg; joints [32.463, -45.843, 104.742, -143.584, 64.757, 163.522] to (-213.68, 106.78, -20) mm, rotated rx 180 ry 0 rz 0.01 deg; joints [32.514, -46.025, 105.13, -143.588, 64.937, 163.633]
  MoveL 1283 to (-179.83, 106.78, -20) mm, rotated rx -180 ry 0 rz 0.01 deg; joints [33.229, -47.252, 107.726, -143.209, 66.251, 164.213]
  MoveC 1284 to (-175.59, 107.91, -20) mm, rotated rx -180 ry 0 rz 0.01 deg; joints [33.359, -47.377, 107.99, -143.111, 66.4, 164.248] to (-172.47, 111.02, -20) mm, rotated rx 180 ry 0 rz 0.01 deg; joints [33.528, -47.418, 108.07, -142.944, 66.482, 164.202]
  MoveC 1285 to (-170.06, 115.13, -20) mm, rotated rx -180 ry 0 rz 0.01 deg; joints [33.716, -47.41, 108.046, -142.745, 66.524, 164.111] to (-167.6, 119.21, -20) mm, rotated rx -180 ry 0 rz 0.01 deg; joints [33.904, -47.404, 108.026, -142.546, 66.569, 164.022]
  MoveC 1286 to (-165.03, 123.23, -20) mm, rotated rx 180 ry 0 rz 0.01 deg; joints [34.091, -47.403, 108.016, -142.348, 66.618, 163.937] to (-162.31, 127.14, -20) mm, rotated rx 180 ry 0 rz 0.01 deg; joints [34.279, -47.409, 108.021, -142.153, 66.674, 163.857]
  MoveC 1287 to (-162.2, 129.16, -20) mm, rotated rx 180 ry 0 rz 0.01 deg; joints [34.347, -47.366, 107.926, -142.069, 66.654, 163.793] to (-164.01, 130.08, -20) mm, rotated rx 180 ry 0 rz 0.01 deg; joints [34.337, -47.281, 107.745, -142.054, 66.574, 163.733]
  MoveC 1288 to (-167.65, 129.69, -20) mm, rotated rx 180 ry 0 rz 0.01 deg; joints [34.244, -47.161, 107.492, -142.115, 66.441, 163.683] to (-171.3, 129.28, -20) mm, rotated rx 180 ry 0 rz 0.01 deg; joints [34.15, -47.042, 107.24, -142.176, 66.307, 163.634]
  MoveC 1289 to (-174.95, 128.97, -20) mm, rotated rx 180 ry 0 rz 0.01 deg; joints [34.06, -46.919, 106.981, -142.234, 66.172, 163.582] to (-178.62, 128.86, -20) mm, rotated rx -180 ry 0 rz 0.01 deg; joints [33.976, -46.791, 106.709, -142.282, 66.033, 163.522]
  MoveL 1290 to (-192.66, 128.86, -20) mm, rotated rx -180 ry 0 rz 0.01 deg; joints [33.672, -46.286, 105.641, -142.444, 65.494, 163.278]
  MoveC 1291 to (-195.95, 129.86, -20) mm, rotated rx -180 ry 0 rz 0.01 deg; joints [33.634, -46.144, 105.339, -142.439, 65.355, 163.188] to (-198.13, 132.51, -20) mm, rotated rx 180 ry 0 rz 0.01 deg; joints [33.672, -46.003, 105.036, -142.354, 65.239, 163.062]
  MoveC 1292 to (-200.31, 135.16, -20) mm, rotated rx 180 ry 0 rz 0.01 deg; joints [33.711, -45.862, 104.733, -142.268, 65.122, 162.936] to (-203.6, 136.15, -20) mm, rotated rx 180 ry 0 rz 0.01 deg; joints [33.673, -45.718, 104.428, -142.262, 64.983, 162.844]
  MoveL 1293 to (-214.9, 136.15, -20) mm, rotated rx -180 ry 0 rz 0.01 deg; joints [33.434, -45.303, 103.552, -142.379, 64.542, 162.642]
  MoveC 1294 to (-223.13, 136.48, -20) mm, rotated rx 180 ry 0 rz 0.01 deg; joints [33.272, -44.989, 102.89, -142.448, 64.214, 162.482] to (-231.31, 137.45, -20) mm, rotated rx -180 ry 0 rz 0.01 deg; joints [33.133, -44.659, 102.195, -142.485, 63.879, 162.3]
  MoveC 1295 to (-239.44, 138.81, -20) mm, rotated rx -180 ry 0 rz 0.01 deg; joints [33.009, -44.32, 101.479, -142.503, 63.539, 162.103] to (-247.53, 140.32, -20) mm, rotated rx 180 ry 0 rz 0.01 deg; joints [32.891, -43.976, 100.753, -142.51, 63.197, 161.9]
  MoveC 1296 to (-249.26, 139.53, -20) mm, rotated rx 180 ry 0 rz 0.01 deg; joints [32.831, -43.928, 100.655, -142.558, 63.137, 161.894] to (-249.09, 137.64, -20) mm, rotated rx 180 ry 0 rz 0.01 deg; joints [32.776, -43.98, 100.767, -142.635, 63.166, 161.963]
  MoveC 1297 to (-243.73, 131.29, -20) mm, rotated rx 180 ry 0 rz 0.01 deg; joints [32.684, -44.335, 101.524, -142.854, 63.456, 162.28] to (-238.53, 124.81, -20) mm, rotated rx 180 ry 0 rz 0.01 deg; joints [32.584, -44.684, 102.269, -143.079, 63.74, 162.594]
  MoveC 1298 to (-233.64, 118.08, -20) mm, rotated rx -180 ry 0 rz 0.01 deg; joints [32.469, -45.024, 102.998, -143.314, 64.014, 162.908] to (-229.24, 111.03, -20) mm, rotated rx 180 ry 0 rz 0.01 deg; joints [32.332, -45.351, 103.699, -143.567, 64.272, 163.22]
  MoveC 1299 to (-228.22, 109.2, -20) mm, rotated rx -180 ry 0 rz 0.01 deg; joints [32.294, -45.431, 103.87, -143.633, 64.334, 163.299] to (-227.27, 107.34, -20) mm, rotated rx -180 ry 0 rz 0.01 deg; joints [32.253, -45.509, 104.038, -143.702, 64.394, 163.377]
  MoveC 1300 to (-226.31, 105.48, -20) mm, rotated rx 180 ry 0 rz 0.01 deg; joints [32.212, -45.587, 104.206, -143.77, 64.454, 163.455] to (-225.29, 103.65, -20) mm, rotated rx 180 ry 0 rz 0.01 deg; joints [32.174, -45.666, 104.376, -143.836, 64.515, 163.532]
  MoveC 1301 to (-222.18, 100.54, -20) mm, rotated rx -180 ry 0 rz 0.01 deg; joints [32.136, -45.851, 104.773, -143.935, 64.675, 163.688] to (-217.94, 99.4, -20) mm, rotated rx -180 ry 0 rz 0.01 deg; joints [32.186, -46.034, 105.161, -143.94, 64.856, 163.799]
  MoveL 1302 to (-175.58, 99.4, -20) mm, rotated rx 180 ry 0 rz 0.01 deg; joints [33.078, -47.568, 108.41, -143.464, 66.502, 164.518]
  MoveC 1303 to (-171.33, 100.54, -20) mm, rotated rx 180 ry 0 rz 0.01 deg; joints [33.207, -47.693, 108.674, -143.364, 66.651, 164.553] to (-168.22, 103.65, -20) mm, rotated rx -180 ry 0 rz 0.01 deg; joints [33.378, -47.734, 108.755, -143.197, 66.733, 164.507]
  MoveC 1304 to (-167.14, 105.59, -20) mm, rotated rx -180 ry 0 rz 0.01 deg; joints [33.466, -47.728, 108.74, -143.103, 66.75, 164.463] to (-166.12, 107.56, -20) mm, rotated rx -180 ry 0 rz 0.01 deg; joints [33.553, -47.72, 108.719, -143.009, 66.765, 164.418]
  MoveC 1305 to (-165.1, 109.53, -20) mm, rotated rx 180 ry 0 rz 0.01 deg; joints [33.64, -47.712, 108.697, -142.914, 66.78, 164.373] to (-164.02, 111.47, -20) mm, rotated rx -180 ry 0 rz 0.01 deg; joints [33.728, -47.706, 108.681, -142.821, 66.798, 164.329]
  MoveC 1306 to (-159.67, 118.42, -20) mm, rotated rx 180 ry 0 rz 0.01 deg; joints [34.052, -47.701, 108.658, -142.479, 66.879, 164.181] to (-154.84, 125.04, -20) mm, rotated rx 180 ry 0 rz 0.01 deg; joints [34.377, -47.719, 108.683, -142.144, 66.981, 164.05]
  MoveC 1307 to (-149.7, 131.41, -20) mm, rotated rx 180 ry 0 rz 0.01 deg; joints [34.7, -47.751, 108.739, -141.815, 67.097, 163.932] to (-144.39, 137.65, -20) mm, rotated rx 180 ry 0 rz 0.01 deg; joints [35.023, -47.79, 108.81, -141.489, 67.219, 163.821]
  MoveC 1308 to (-144.2, 139.54, -20) mm, rotated rx 180 ry 0 rz 0.01 deg; joints [35.089, -47.752, 108.727, -141.409, 67.203, 163.763] to (-145.93, 140.33, -20) mm, rotated rx -180 ry 0 rz 0.01 deg; joints [35.075, -47.674, 108.559, -141.4, 67.129, 163.708]
  MoveC 1309 to (-154.04, 138.82, -20) mm, rotated rx 180 ry 0 rz 0.01 deg; joints [34.843, -47.427, 108.038, -141.568, 66.844, 163.619] to (-162.17, 137.45, -20) mm, rotated rx 180 ry 0 rz 0.01 deg; joints [34.616, -47.174, 107.504, -141.728, 66.555, 163.525]
  MoveC 1310 to (-170.37, 136.48, -20) mm, rotated rx -180 ry 0 rz 0.01 deg; joints [34.403, -46.907, 106.941, -141.869, 66.256, 163.415] to (-178.62, 136.15, -20) mm, rotated rx -180 ry 0 rz 0.01 deg; joints [34.211, -46.621, 106.337, -141.981, 65.946, 163.283]
  MoveL 1311 to (-203.6, 136.15, -20) mm, rotated rx 180 ry 0 rz 0.01 deg; joints [33.673, -45.718, 104.428, -142.262, 64.983, 162.844]
  MoveC 1312 to (-206.7, 137.09, -20) mm, rotated rx 180 ry 0 rz 0.01 deg; joints [33.637, -45.583, 104.141, -142.256, 64.851, 162.758] to (-208.75, 139.59, -20) mm, rotated rx 180 ry 0 rz 0.01 deg; joints [33.673, -45.448, 103.853, -142.174, 64.741, 162.637]
  MoveC 1313 to (-210.81, 142.09, -20) mm, rotated rx -180 ry 0 rz 0.01 deg; joints [33.708, -45.313, 103.564, -142.092, 64.631, 162.516] to (-213.9, 143.02, -20) mm, rotated rx 180 ry 0 rz 0.01 deg; joints [33.673, -45.177, 103.274, -142.085, 64.499, 162.429]
  MoveL 1314 to (-214.9, 143.02, -20) mm, rotated rx -180 ry 0 rz 0.01 deg; joints [33.652, -45.14, 103.197, -142.095, 64.46, 162.411]
  MoveC 1315 to (-230.2, 143.85, -20) mm, rotated rx 180 ry 0 rz 0.01 deg; joints [33.358, -44.549, 101.951, -142.208, 63.847, 162.102] to (-245.33, 146.33, -20) mm, rotated rx 180 ry 0 rz 0.01 deg; joints [33.125, -43.916, 100.617, -142.24, 63.215, 161.734]
  MoveC 1316 to (-260.13, 150.28, -20) mm, rotated rx -180 ry 0 rz 0.01 deg; joints [32.948, -43.251, 99.214, -142.196, 62.572, 161.314] to (-274.52, 155.53, -20) mm, rotated rx -180 ry 0 rz 0.01 deg; joints [32.822, -42.559, 97.756, -142.081, 61.923, 160.845]
  MoveC 1317 to (-276.08, 155, -20) mm, rotated rx 180 ry 0 rz 0.01 deg; joints [32.775, -42.511, 97.655, -142.114, 61.866, 160.833] to (-275.75, 153.39, -20) mm, rotated rx 180 ry 0 rz 0.01 deg; joints [32.732, -42.563, 97.768, -142.18, 61.898, 160.897]
  MoveC 1318 to (-266.78, 146.05, -20) mm, rotated rx 180 ry 0 rz 0.01 deg; joints [32.683, -43.094, 98.893, -142.424, 62.351, 161.333] to (-258.39, 138.07, -20) mm, rotated rx -180 ry 0 rz 0.01 deg; joints [32.602, -43.612, 99.993, -142.694, 62.786, 161.772]
  MoveC 1319 to (-250.57, 129.52, -20) mm, rotated rx -180 ry 0 rz 0.01 deg; joints [32.49, -44.116, 101.066, -142.988, 63.202, 162.213] to (-243.33, 120.47, -20) mm, rotated rx 180 ry 0 rz 0.01 deg; joints [32.348, -44.603, 102.106, -143.303, 63.599, 162.653]
  MoveC 1320 to (-241.11, 117.37, -20) mm, rotated rx 180 ry 0 rz 0.01 deg; joints [32.294, -44.759, 102.44, -143.413, 63.724, 162.797] to (-239.02, 114.19, -20) mm, rotated rx 180 ry 0 rz 0.01 deg; joints [32.235, -44.911, 102.766, -143.527, 63.845, 162.941]
  MoveC 1321 to (-237.02, 110.95, -20) mm, rotated rx 180 ry 0 rz 0.01 deg; joints [32.171, -45.061, 103.087, -143.644, 63.963, 163.084] to (-235.09, 107.67, -20) mm, rotated rx -180 ry 0 rz 0.01 deg; joints [32.104, -45.208, 103.404, -143.763, 64.079, 163.227]
  MoveC 1322 to (-233.59, 104.97, -20) mm, rotated rx -180 ry 0 rz 0.01 deg; joints [32.048, -45.326, 103.657, -143.862, 64.17, 163.343] to (-232.17, 102.22, -20) mm, rotated rx -180 ry 0 rz 0.01 deg; joints [31.987, -45.441, 103.904, -143.963, 64.259, 163.458]
  MoveC 1323 to (-230.76, 99.48, -20) mm, rotated rx 180 ry 0 rz 0.01 deg; joints [31.927, -45.555, 104.151, -144.064, 64.347, 163.572] to (-229.26, 96.78, -20) mm, rotated rx -180 ry 0 rz 0.01 deg; joints [31.87, -45.672, 104.402, -144.163, 64.438, 163.687]
  MoveC 1324 to (-226.15, 93.67, -20) mm, rotated rx 180 ry 0 rz 0.01 deg; joints [31.831, -45.857, 104.798, -144.262, 64.598, 163.841] to (-221.91, 92.53, -20) mm, rotated rx 180 ry 0 rz 0.01 deg; joints [31.88, -46.04, 105.186, -144.267, 64.78, 163.951]
  MoveL 1325 to (-171.61, 92.53, -20) mm, rotated rx 180 ry 0 rz 0.01 deg; joints [32.935, -47.86, 109.044, -143.7, 66.736, 164.8]
  MoveC 1326 to (-167.36, 93.67, -20) mm, rotated rx 180 ry 0 rz 0.01 deg; joints [33.065, -47.985, 109.308, -143.6, 66.885, 164.834] to (-164.25, 96.78, -20) mm, rotated rx 180 ry 0 rz 0.01 deg; joints [33.236, -48.026, 109.388, -143.432, 66.966, 164.788]
  MoveC 1327 to (-162.69, 99.58, -20) mm, rotated rx -180 ry 0 rz 0.01 deg; joints [33.364, -48.019, 109.368, -143.295, 66.992, 164.726] to (-161.22, 102.44, -20) mm, rotated rx -180 ry 0 rz 0.01 deg; joints [33.491, -48.007, 109.338, -143.158, 67.013, 164.661]
  MoveC 1328 to (-159.74, 105.29, -20) mm, rotated rx -180 ry 0 rz 0.01 deg; joints [33.618, -47.995, 109.307, -143.022, 67.035, 164.596] to (-158.18, 108.09, -20) mm, rotated rx 180 ry 0 rz 0.01 deg; joints [33.745, -47.987, 109.284, -142.885, 67.06, 164.533]
  MoveC 1329 to (-149.84, 120.91, -20) mm, rotated rx -180 ry 0 rz 0.01 deg; joints [34.354, -47.987, 109.261, -142.248, 67.219, 164.266] to (-140.18, 132.76, -20) mm, rotated rx 180 ry 0 rz 0.01 deg; joints [34.96, -48.048, 109.369, -141.633, 67.435, 164.049]
  MoveC 1330 to (-129.41, 143.6, -20) mm, rotated rx -180 ry 0 rz 0.01 deg; joints [35.561, -48.164, 109.596, -141.041, 67.702, 163.881] to (-117.71, 153.43, -20) mm, rotated rx 180 ry 0 rz 0.01 deg; joints [36.153, -48.329, 109.929, -140.475, 68.01, 163.759]
  MoveC 1331 to (-117.39, 155.04, -20) mm, rotated rx -180 ry 0 rz 0.01 deg; joints [36.212, -48.302, 109.867, -140.405, 68.002, 163.712] to (-118.95, 155.56, -20) mm, rotated rx -180 ry 0 rz 0.01 deg; joints [36.192, -48.237, 109.728, -140.407, 67.939, 163.669]
  MoveC 1332 to (-129.3, 151.62, -20) mm, rotated rx 180 ry 0 rz 0.01 deg; joints [35.823, -47.979, 109.187, -140.713, 67.608, 163.623] to (-139.9, 148.43, -20) mm, rotated rx 180 ry 0 rz 0.01 deg; joints [35.475, -47.691, 108.581, -140.989, 67.255, 163.547]
  MoveC 1333 to (-150.7, 145.97, -20) mm, rotated rx -180 ry 0 rz 0.01 deg; joints [35.149, -47.375, 107.916, -141.232, 66.883, 163.443] to (-161.62, 144.16, -20) mm, rotated rx 180 ry 0 rz 0.01 deg; joints [34.845, -47.036, 107.199, -141.446, 66.494, 163.315]
  MoveC 1334 to (-170.1, 143.31, -20) mm, rotated rx -180 ry 0 rz 0.01 deg; joints [34.629, -46.756, 106.609, -141.585, 66.184, 163.196] to (-178.62, 143.02, -20) mm, rotated rx 180 ry 0 rz 0.01 deg; joints [34.432, -46.46, 105.983, -141.699, 65.863, 163.057]
  MoveL 1335 to (-213.9, 143.02, -20) mm, rotated rx -180 ry 0 rz 0.01 deg; joints [33.673, -45.177, 103.274, -142.085, 64.499, 162.429]
  MoveC 1336 to (-216.88, 143.93, -20) mm, rotated rx -180 ry 0 rz 0.01 deg; joints [33.639, -45.045, 102.995, -142.077, 64.372, 162.344] to (-218.85, 146.35, -20) mm, rotated rx -180 ry 0 rz 0.01 deg; joints [33.674, -44.914, 102.715, -141.996, 64.266, 162.226]
  MoveC 1337 to (-220.76, 148.78, -20) mm, rotated rx -180 ry 0 rz 0.01 deg; joints [33.71, -44.784, 102.438, -141.914, 64.162, 162.108] to (-223.68, 149.82, -20) mm, rotated rx 180 ry 0 rz 0.01 deg; joints [33.682, -44.65, 102.154, -141.899, 64.034, 162.019]
  MoveC 1338 to (-236.97, 151.3, -20) mm, rotated rx 180 ry 0 rz 0.01 deg; joints [33.452, -44.114, 101.024, -141.96, 63.49, 161.72] to (-250.06, 154.05, -20) mm, rotated rx 180 ry 0 rz 0.01 deg; joints [33.269, -43.548, 99.83, -141.958, 62.934, 161.376]
  MoveC 1339 to (-266.96, 159.49, -20) mm, rotated rx -180 ry 0 rz 0.01 deg; joints [33.095, -42.758, 98.166, -141.861, 62.186, 160.854] to (-283.14, 166.82, -20) mm, rotated rx -180 ry 0 rz 0.01 deg; joints [32.997, -41.937, 96.435, -141.663, 61.436, 160.266]
  MoveC 1340 to (-285.4, 166.75, -20) mm, rotated rx -180 ry 0 rz 0.01 deg; joints [32.95, -41.848, 96.25, -141.68, 61.344, 160.222] to (-286.51, 164.78, -20) mm, rotated rx -180 ry 0 rz 0.01 deg; joints [32.869, -41.853, 96.264, -141.77, 61.321, 160.271]
  MoveL 1341 to (-286.5, 156.62, -20) mm, rotated rx -180 ry 0 rz 0.01 deg; joints [32.619, -42.056, 96.702, -142.115, 61.417, 160.566]
  MoveC 1342 to (-285.74, 153.49, -20) mm, rotated rx -180 ry 0 rz 0.01 deg; joints [32.538, -42.164, 96.933, -142.242, 61.485, 160.693] to (-283.63, 151.06, -20) mm, rotated rx 180 ry 0 rz 0.01 deg; joints [32.505, -42.308, 97.238, -142.331, 61.601, 160.823]
  MoveC 1343 to (-271.09, 141.19, -20) mm, rotated rx -180 ry 0 rz 0.01 deg; joints [32.446, -43.043, 98.794, -142.66, 62.232, 161.419] to (-259.61, 130.1, -20) mm, rotated rx -180 ry 0 rz 0.01 deg; joints [32.327, -43.754, 100.305, -143.038, 62.83, 162.024]
  MoveC 1344 to (-249.39, 117.83, -20) mm, rotated rx -180 ry 0 rz 0.01 deg; joints [32.142, -44.434, 101.755, -143.467, 63.386, 162.631] to (-240.63, 104.47, -20) mm, rotated rx 180 ry 0 rz 0.01 deg; joints [31.889, -45.072, 103.122, -143.949, 63.894, 163.234]
  MoveC 1345 to (-238.68, 100.95, -20) mm, rotated rx -180 ry 0 rz 0.01 deg; joints [31.815, -45.225, 103.452, -144.078, 64.014, 163.385] to (-236.83, 97.36, -20) mm, rotated rx -180 ry 0 rz 0.01 deg; joints [31.736, -45.375, 103.774, -144.211, 64.129, 163.535]
  MoveC 1346 to (-234.98, 93.78, -20) mm, rotated rx 180 ry 0 rz 0.01 deg; joints [31.656, -45.524, 104.096, -144.344, 64.245, 163.684] to (-233.03, 90.26, -20) mm, rotated rx -180 ry 0 rz 0.01 deg; joints [31.581, -45.676, 104.422, -144.473, 64.364, 163.832]
  MoveC 1347 to (-229.92, 87.15, -20) mm, rotated rx -180 ry 0 rz 0.01 deg; joints [31.541, -45.861, 104.818, -144.573, 64.524, 163.986] to (-225.68, 86.01, -20) mm, rotated rx -180 ry 0 rz 0.01 deg; joints [31.59, -46.044, 105.207, -144.578, 64.706, 164.096]
  MoveL 1348 to (-167.85, 86.01, -20) mm, rotated rx 180 ry 0 rz 0.01 deg; joints [32.798, -48.135, 109.642, -143.924, 66.958, 165.064]
  MoveC 1349 to (-163.6, 87.15, -20) mm, rotated rx 180 ry 0 rz 0.01 deg; joints [32.929, -48.26, 109.905, -143.823, 67.106, 165.099] to (-160.49, 90.26, -20) mm, rotated rx -180 ry 0 rz 0.01 deg; joints [33.101, -48.301, 109.987, -143.654, 67.187, 165.053]
  MoveC 1350 to (-158.47, 93.89, -20) mm, rotated rx 180 ry 0 rz 0.01 deg; joints [33.266, -48.292, 109.961, -143.477, 67.22, 164.974] to (-156.56, 97.57, -20) mm, rotated rx 180 ry 0 rz 0.01 deg; joints [33.432, -48.277, 109.922, -143.3, 67.248, 164.89]
  MoveC 1351 to (-154.66, 101.26, -20) mm, rotated rx 180 ry 0 rz 0.01 deg; joints [33.597, -48.262, 109.883, -143.122, 67.275, 164.806] to (-152.63, 104.89, -20) mm, rotated rx 180 ry 0 rz 0.01 deg; joints [33.762, -48.252, 109.854, -142.945, 67.308, 164.726]
  MoveC 1352 to (-143.93, 118.14, -20) mm, rotated rx 180 ry 0 rz 0.01 deg; joints [34.395, -48.255, 109.835, -142.283, 67.474, 164.452] to (-133.78, 130.31, -20) mm, rotated rx 180 ry 0 rz 0.01 deg; joints [35.026, -48.325, 109.962, -141.645, 67.703, 164.234]
  MoveC 1353 to (-122.37, 141.3, -20) mm, rotated rx 180 ry 0 rz 0.01 deg; joints [35.65, -48.458, 110.224, -141.035, 67.989, 164.073] to (-109.9, 151.07, -20) mm, rotated rx -180 ry 0 rz 0.01 deg; joints [36.261, -48.648, 110.611, -140.456, 68.324, 163.966]
  MoveC 1354 to (-107.77, 153.5, -20) mm, rotated rx 180 ry 0 rz 0.01 deg; joints [36.391, -48.661, 110.635, -140.326, 68.371, 163.923] to (-107.01, 156.64, -20) mm, rotated rx -180 ry 0 rz 0.01 deg; joints [36.51, -48.612, 110.525, -140.188, 68.36, 163.834]
  MoveL 1355 to (-107.01, 164.77, -20) mm, rotated rx -180 ry 0 rz 0.01 deg; joints [36.772, -48.417, 110.095, -139.86, 68.259, 163.57]
  MoveC 1356 to (-108.12, 166.73, -20) mm, rotated rx -180 ry 0 rz 0.01 deg; joints [36.808, -48.333, 109.912, -139.797, 68.195, 163.487] to (-110.37, 166.8, -20) mm, rotated rx -180 ry 0 rz 0.01 deg; joints [36.756, -48.256, 109.748, -139.828, 68.112, 163.447]
  MoveC 1357 to (-122.79, 160.99, -20) mm, rotated rx 180 ry 0 rz 0.01 deg; joints [36.276, -47.976, 109.165, -140.242, 67.731, 163.427] to (-135.72, 156.41, -20) mm, rotated rx -180 ry 0 rz 0.01 deg; joints [35.828, -47.645, 108.469, -140.607, 67.312, 163.357]
  MoveC 1358 to (-148.99, 152.98, -20) mm, rotated rx 180 ry 0 rz 0.01 deg; joints [35.413, -47.268, 107.676, -140.924, 66.861, 163.242] to (-162.49, 150.62, -20) mm, rotated rx 180 ry 0 rz 0.01 deg; joints [35.033, -46.852, 106.798, -141.192, 66.383, 163.087]
  MoveC 1359 to (-170.54, 149.81, -20) mm, rotated rx -180 ry 0 rz 0.01 deg; joints [34.827, -46.587, 106.239, -141.324, 66.089, 162.974] to (-178.62, 149.54, -20) mm, rotated rx -180 ry 0 rz 0.01 deg; joints [34.64, -46.305, 105.644, -141.431, 65.785, 162.841]
  MoveL 1360 to (-214.9, 149.54, -20) mm, rotated rx -180 ry 0 rz 0.01 deg; joints [33.858, -44.984, 102.857, -141.825, 64.383, 162.19]
  MoveC 1361 to (-219.29, 149.61, -20) mm, rotated rx 180 ry 0 rz 0.01 deg; joints [33.767, -44.819, 102.51, -141.865, 64.21, 162.107] to (-223.68, 149.82, -20) mm, rotated rx 180 ry 0 rz 0.01 deg; joints [33.682, -44.65, 102.154, -141.899, 64.034, 162.019]
  MoveC 1362 to (-227.3, 151.19, -20) mm, rotated rx 180 ry 0 rz 0.01 deg; joints [33.649, -44.482, 101.797, -141.877, 63.875, 161.905] to (-229.54, 154.35, -20) mm, rotated rx 180 ry 0 rz 0.01 deg; joints [33.701, -44.321, 101.454, -141.766, 63.749, 161.754]
  MoveC 1363 to (-231.69, 157.53, -20) mm, rotated rx -180 ry 0 rz 0.01 deg; joints [33.756, -44.162, 101.115, -141.654, 63.626, 161.604] to (-235.2, 159.11, -20) mm, rotated rx 180 ry 0 rz 0.01 deg; joints [33.732, -43.991, 100.753, -141.62, 63.468, 161.483]
  MoveC 1364 to (-257.17, 164.18, -20) mm, rotated rx 180 ry 0 rz 0.01 deg; joints [33.437, -43.024, 98.715, -141.591, 62.528, 160.881] to (-278.03, 172.73, -20) mm, rotated rx 180 ry 0 rz 0.01 deg; joints [33.279, -41.991, 96.539, -141.381, 61.577, 160.155]
  MoveC 1365 to (-281.48, 174.62, -20) mm, rotated rx 180 ry 0 rz 0.01 deg; joints [33.267, -41.806, 96.149, -141.324, 61.413, 160.016] to (-284.78, 176.74, -20) mm, rotated rx -180 ry 0 rz 0.01 deg; joints [33.266, -41.62, 95.757, -141.255, 61.251, 159.869]
  MoveC 1366 to (-288.03, 178.95, -20) mm, rotated rx 180 ry 0 rz 0.01 deg; joints [33.268, -41.433, 95.364, -141.181, 61.091, 159.72] to (-291.31, 181.11, -20) mm, rotated rx -180 ry 0 rz 0.01 deg; joints [33.269, -41.246, 94.969, -141.109, 60.929, 159.571]
  MoveC 1367 to (-293.48, 181.19, -20) mm, rotated rx 180 ry 0 rz 0.01 deg; joints [33.228, -41.156, 94.781, -141.117, 60.838, 159.522] to (-294.59, 179.32, -20) mm, rotated rx 180 ry 0 rz 0.01 deg; joints [33.15, -41.159, 94.79, -141.203, 60.814, 159.568]
  MoveL 1368 to (-294.58, 153.81, -20) mm, rotated rx -180 ry 0 rz 0.01 deg; joints [32.375, -41.802, 96.175, -142.283, 61.115, 160.502]
  MoveC 1369 to (-293.49, 149.38, -20) mm, rotated rx -180 ry 0 rz 0.01 deg; joints [32.261, -41.955, 96.502, -142.464, 61.212, 160.684] to (-290.45, 145.97, -20) mm, rotated rx -180 ry 0 rz 0.01 deg; joints [32.215, -42.16, 96.937, -142.59, 61.378, 160.868]
  MoveC 1370 to (-280.55, 138.56, -20) mm, rotated rx -180 ry 0 rz 0.01 deg; joints [32.178, -42.734, 98.151, -142.838, 61.874, 161.327] to (-271.33, 130.31, -20) mm, rotated rx -180 ry 0 rz 0.01 deg; joints [32.101, -43.293, 99.338, -143.119, 62.35, 161.794]
  MoveC 1371 to (-262.81, 121.34, -20) mm, rotated rx -180 ry 0 rz 0.01 deg; joints [31.987, -43.836, 100.492, -143.431, 62.802, 162.263] to (-255.03, 111.73, -20) mm, rotated rx 180 ry 0 rz 0.01 deg; joints [31.835, -44.358, 101.607, -143.771, 63.23, 162.732]
  MoveC 1372 to (-251.15, 106.2, -20) mm, rotated rx -180 ry 0 rz 0.01 deg; joints [31.735, -44.633, 102.195, -143.97, 63.451, 162.988] to (-247.6, 100.45, -20) mm, rotated rx 180 ry 0 rz 0.01 deg; joints [31.621, -44.898, 102.764, -144.18, 63.661, 163.242]
  MoveC 1373 to (-245.07, 95.92, -20) mm, rotated rx 180 ry 0 rz 0.01 deg; joints [31.524, -45.096, 103.189, -144.348, 63.816, 163.436] to (-242.65, 91.32, -20) mm, rotated rx -180 ry 0 rz 0.01 deg; joints [31.423, -45.29, 103.607, -144.519, 63.966, 163.629]
  MoveC 1374 to (-240.23, 86.71, -20) mm, rotated rx -180 ry 0 rz 0.01 deg; joints [31.321, -45.483, 104.022, -144.69, 64.117, 163.821] to (-237.7, 82.18, -20) mm, rotated rx -180 ry 0 rz 0.01 deg; joints [31.223, -45.678, 104.443, -144.856, 64.271, 164.012]
  MoveC 1375 to (-234.59, 79.07, -20) mm, rotated rx -180 ry 0 rz 0.01 deg; joints [31.182, -45.863, 104.838, -144.957, 64.432, 164.165] to (-230.35, 77.93, -20) mm, rotated rx -180 ry 0 rz 0.01 deg; joints [31.23, -46.046, 105.227, -144.964, 64.615, 164.274]
  MoveL 1376 to (-163.19, 77.93, -20) mm, rotated rx 180 ry 0 rz 0.01 deg; joints [32.627, -48.474, 110.379, -144.202, 67.232, 165.389]
  MoveC 1377 to (-158.94, 79.07, -20) mm, rotated rx 180 ry 0 rz 0.01 deg; joints [32.758, -48.598, 110.641, -144.099, 67.38, 165.423] to (-155.83, 82.18, -20) mm, rotated rx 180 ry 0 rz 0.01 deg; joints [32.931, -48.639, 110.723, -143.929, 67.461, 165.378]
  MoveC 1378 to (-153.23, 86.82, -20) mm, rotated rx -180 ry 0 rz 0.01 deg; joints [33.144, -48.629, 110.693, -143.702, 67.504, 165.278] to (-150.74, 91.52, -20) mm, rotated rx 180 ry 0 rz 0.01 deg; joints [33.357, -48.613, 110.649, -143.474, 67.541, 165.173]
  MoveC 1379 to (-148.26, 96.22, -20) mm, rotated rx 180 ry 0 rz 0.01 deg; joints [33.57, -48.596, 110.603, -143.246, 67.577, 165.068] to (-145.66, 100.86, -20) mm, rotated rx 180 ry 0 rz 0.01 deg; joints [33.783, -48.583, 110.567, -143.019, 67.619, 164.966]
  MoveC 1380 to (-137.06, 113.9, -20) mm, rotated rx -180 ry 0 rz 0.01 deg; joints [34.411, -48.587, 110.551, -142.364, 67.782, 164.699] to (-126.97, 125.83, -20) mm, rotated rx -180 ry 0 rz 0.01 deg; joints [35.036, -48.66, 110.684, -141.733, 68.009, 164.489]
  MoveC 1381 to (-115.6, 136.53, -20) mm, rotated rx 180 ry 0 rz 0.01 deg; joints [35.653, -48.798, 110.957, -141.131, 68.295, 164.337] to (-103.12, 145.92, -20) mm, rotated rx -180 ry 0 rz 0.01 deg; joints [36.255, -48.996, 111.362, -140.563, 68.633, 164.244]
  MoveC 1382 to (-100.04, 149.33, -20) mm, rotated rx 180 ry 0 rz 0.01 deg; joints [36.44, -49.018, 111.403, -140.378, 68.702, 164.186] to (-98.93, 153.79, -20) mm, rotated rx 180 ry 0 rz 0.01 deg; joints [36.612, -48.949, 111.248, -140.181, 68.687, 164.061]
  MoveL 1383 to (-98.93, 179.33, -20) mm, rotated rx -180 ry 0 rz 0.01 deg; joints [37.432, -48.332, 109.888, -139.153, 68.37, 163.228]
  MoveC 1384 to (-100.03, 181.19, -20) mm, rotated rx 180 ry 0 rz 0.01 deg; joints [37.464, -48.25, 109.709, -139.095, 68.307, 163.148] to (-102.2, 181.11, -20) mm, rotated rx 180 ry 0 rz 0.01 deg; joints [37.409, -48.18, 109.56, -139.131, 68.23, 163.114]
  MoveC 1385 to (-109.98, 176.31, -20) mm, rotated rx 180 ry 0 rz 0.01 deg; joints [37.069, -48.037, 109.266, -139.439, 68.009, 163.14] to (-117.96, 171.85, -20) mm, rotated rx 180 ry 0 rz 0.01 deg; joints [36.737, -47.877, 108.935, -139.734, 67.774, 163.152]
  MoveC 1386 to (-126.22, 167.91, -20) mm, rotated rx -180 ry 0 rz 0.01 deg; joints [36.416, -47.693, 108.55, -140.01, 67.521, 163.141] to (-134.79, 164.69, -20) mm, rotated rx 180 ry 0 rz 0.01 deg; joints [36.114, -47.477, 108.099, -140.258, 67.245, 163.1]
  MoveC 1387 to (-154.43, 159.86, -20) mm, rotated rx -180 ry 0 rz 0.01 deg; joints [35.509, -46.914, 106.912, -140.713, 66.574, 162.921] to (-174.56, 157.99, -20) mm, rotated rx -180 ry 0 rz 0.01 deg; joints [34.998, -46.247, 105.507, -141.037, 65.837, 162.63]
  MoveL 1388 to (-214.9, 157.62, -20) mm, rotated rx 180 ry 0 rz 0.01 deg; joints [34.111, -44.789, 102.432, -141.49, 64.287, 161.914]
  MoveC 1389 to (-225.08, 158, -20) mm, rotated rx 180 ry 0 rz 0.01 deg; joints [33.908, -44.4, 101.614, -141.573, 63.882, 161.712] to (-235.2, 159.11, -20) mm, rotated rx -180 ry 0 rz 0.01 deg; joints [33.732, -43.991, 100.753, -141.62, 63.468, 161.483]
  MoveC 1390 to (-238.61, 160.73, -20) mm, rotated rx 180 ry 0 rz 0.01 deg; joints [33.711, -43.822, 100.395, -141.582, 63.313, 161.361] to (-240.52, 163.99, -20) mm, rotated rx 180 ry 0 rz 0.01 deg; joints [33.773, -43.669, 100.069, -141.464, 63.199, 161.211]
  MoveC 1391 to (-242.34, 167.26, -20) mm, rotated rx 180 ry 0 rz 0.01 deg; joints [33.836, -43.519, 99.747, -141.343, 63.087, 161.06] to (-245.61, 169.1, -20) mm, rotated rx 180 ry 0 rz 0.01 deg; joints [33.825, -43.348, 99.386, -141.294, 62.934, 160.932]
  MoveC 1392 to (-260.38, 173.55, -20) mm, rotated rx 180 ry 0 rz 0.01 deg; joints [33.659, -42.665, 97.948, -141.224, 62.287, 160.482] to (-274.53, 179.7, -20) mm, rotated rx 180 ry 0 rz 0.01 deg; joints [33.56, -41.953, 96.449, -141.065, 61.638, 159.973]
  MoveC 1393 to (-281.08, 183.31, -20) mm, rotated rx 180 ry 0 rz 0.01 deg; joints [33.538, -41.6, 95.705, -140.955, 61.326, 159.704] to (-287.33, 187.43, -20) mm, rotated rx 180 ry 0 rz 0.01 deg; joints [33.537, -41.243, 94.953, -140.819, 61.019, 159.421]
  MoveC 1394 to (-293.36, 191.85, -20) mm, rotated rx -180 ry 0 rz 0.01 deg; joints [33.55, -40.884, 94.197, -140.666, 60.717, 159.126] to (-299.27, 196.42, -20) mm, rotated rx 180 ry 0 rz 0.01 deg; joints [33.569, -40.523, 93.437, -140.502, 60.416, 158.825]
  MoveC 1395 to (-301.34, 196.65, -20) mm, rotated rx 180 ry 0 rz 0.01 deg; joints [33.536, -40.433, 93.248, -140.502, 60.327, 158.771] to (-302.44, 194.89, -20) mm, rotated rx 180 ry 0 rz 0.01 deg; joints [33.462, -40.434, 93.253, -140.582, 60.302, 158.814]
  MoveL 1396 to (-302.44, 149.18, -20) mm, rotated rx -180 ry 0 rz 0.01 deg; joints [32.082, -41.598, 95.757, -142.524, 60.84, 160.509]
  MoveC 1397 to (-301.34, 144.93, -20) mm, rotated rx -180 ry 0 rz 0.01 deg; joints [31.972, -41.747, 96.075, -142.699, 60.936, 160.684] to (-298.33, 141.75, -20) mm, rotated rx -180 ry 0 rz 0.01 deg; joints [31.932, -41.946, 96.498, -142.816, 61.099, 160.86]
  MoveC 1398 to (-287.88, 134.43, -20) mm, rotated rx 180 ry 0 rz 0.01 deg; joints [31.907, -42.542, 97.756, -143.061, 61.62, 161.328] to (-278.22, 126.09, -20) mm, rotated rx 180 ry 0 rz 0.01 deg; joints [31.834, -43.123, 98.987, -143.347, 62.116, 161.807]
  MoveC 1399 to (-269.37, 116.91, -20) mm, rotated rx 180 ry 0 rz 0.01 deg; joints [31.717, -43.684, 100.181, -143.669, 62.586, 162.291] to (-261.31, 107.02, -20) mm, rotated rx -180 ry 0 rz 0.01 deg; joints [31.561, -44.224, 101.333, -144.021, 63.029, 162.775]
  MoveC 1400 to (-257.7, 101.88, -20) mm, rotated rx 180 ry 0 rz 0.01 deg; joints [31.467, -44.48, 101.881, -144.207, 63.236, 163.012] to (-254.41, 96.53, -20) mm, rotated rx 180 ry 0 rz 0.01 deg; joints [31.359, -44.727, 102.41, -144.404, 63.431, 163.249]
  MoveC 1401 to (-251.3, 91.01, -20) mm, rotated rx 180 ry 0 rz 0.01 deg; joints [31.242, -44.969, 102.929, -144.609, 63.621, 163.486] to (-248.32, 85.43, -20) mm, rotated rx -180 ry 0 rz 0.01 deg; joints [31.119, -45.206, 103.439, -144.818, 63.806, 163.721]
  MoveC 1402 to (-245.34, 79.84, -20) mm, rotated rx -180 ry 0 rz 0.01 deg; joints [30.995, -45.441, 103.946, -145.026, 63.991, 163.954] to (-242.23, 74.32, -20) mm, rotated rx -180 ry 0 rz 0.01 deg; joints [30.875, -45.678, 104.457, -145.229, 64.18, 164.185]
  MoveC 1403 to (-239.13, 71.22, -20) mm, rotated rx -180 ry 0 rz 0.01 deg; joints [30.833, -45.862, 104.852, -145.331, 64.341, 164.338] to (-234.89, 70.08, -20) mm, rotated rx 180 ry 0 rz 0.01 deg; joints [30.88, -46.046, 105.242, -145.338, 64.524, 164.446]
  MoveL 1404 to (-158.66, 70.08, -20) mm, rotated rx -180 ry 0 rz 0.01 deg; joints [32.459, -48.8, 111.089, -144.471, 67.499, 165.702]
  MoveC 1405 to (-154.41, 71.22, -20) mm, rotated rx 180 ry 0 rz 0.01 deg; joints [32.59, -48.924, 111.351, -144.367, 67.647, 165.735] to (-151.3, 74.33, -20) mm, rotated rx -180 ry 0 rz 0.01 deg; joints [32.764, -48.966, 111.434, -144.196, 67.727, 165.69]
  MoveL 1406 to (-138.86, 96.93, -20) mm, rotated rx 180 ry 0 rz 0.01 deg; joints [33.804, -48.904, 111.259, -143.089, 67.921, 165.199]
  MoveC 1407 to (-130.1, 110.06, -20) mm, rotated rx 180 ry 0 rz 0.01 deg; joints [34.442, -48.911, 111.249, -142.424, 68.087, 164.933] to (-119.73, 121.97, -20) mm, rotated rx -180 ry 0 rz 0.01 deg; joints [35.077, -48.994, 111.402, -141.786, 68.323, 164.73]
  MoveC 1408 to (-108.01, 132.54, -20) mm, rotated rx -180 ry 0 rz 0.01 deg; joints [35.7, -49.145, 111.704, -141.181, 68.621, 164.589] to (-95.19, 141.73, -20) mm, rotated rx -180 ry 0 rz 0.01 deg; joints [36.309, -49.357, 112.141, -140.611, 68.971, 164.508]
  MoveC 1409 to (-92.17, 144.95, -20) mm, rotated rx 180 ry 0 rz 0.01 deg; joints [36.487, -49.381, 112.187, -140.434, 69.039, 164.455] to (-91.07, 149.22, -20) mm, rotated rx 180 ry 0 rz 0.01 deg; joints [36.653, -49.317, 112.041, -140.244, 69.026, 164.337]
  MoveL 1410 to (-91.07, 194.92, -20) mm, rotated rx 180 ry 0 rz 0.01 deg; joints [38.116, -48.206, 109.591, -138.41, 68.457, 162.843]
  MoveC 1411 to (-92.18, 196.68, -20) mm, rotated rx 180 ry 0 rz 0.01 deg; joints [38.144, -48.125, 109.417, -138.357, 68.396, 162.765] to (-94.25, 196.46, -20) mm, rotated rx -180 ry 0 rz 0.01 deg; joints [38.086, -48.062, 109.284, -138.398, 68.325, 162.738]
  MoveC 1412 to (-101.57, 190.92, -20) mm, rotated rx 180 ry 0 rz 0.01 deg; joints [37.733, -47.957, 109.071, -138.729, 68.131, 162.798] to (-109.11, 185.67, -20) mm, rotated rx 180 ry 0 rz 0.01 deg; joints [37.386, -47.836, 108.822, -139.05, 67.925, 162.844]
  MoveC 1413 to (-116.95, 180.88, -20) mm, rotated rx -180 ry 0 rz 0.01 deg; joints [37.047, -47.69, 108.521, -139.356, 67.7, 162.869] to (-125.16, 176.75, -20) mm, rotated rx -180 ry 0 rz 0.01 deg; joints [36.722, -47.513, 108.153, -139.638, 67.451, 162.866]
  MoveC 1414 to (-146.79, 169.4, -20) mm, rotated rx 180 ry 0 rz 0.01 deg; joints [35.986, -46.949, 106.97, -140.227, 66.743, 162.736] to (-169.43, 166.34, -20) mm, rotated rx 180 ry 0 rz 0.01 deg; joints [35.376, -46.228, 105.451, -140.635, 65.931, 162.441]
  MoveL 1415 to (-214.9, 165.48, -20) mm, rotated rx -180 ry 0 rz 0.01 deg; joints [34.357, -44.597, 102.015, -141.166, 64.193, 161.643]
  MoveC 1416 to (-230.36, 166.39, -20) mm, rotated rx -180 ry 0 rz 0.01 deg; joints [34.058, -43.996, 100.749, -141.274, 63.574, 161.321] to (-245.61, 169.1, -20) mm, rotated rx -180 ry 0 rz 0.01 deg; joints [33.825, -43.348, 99.386, -141.294, 62.934, 160.932]
  MoveC 1417 to (-248.76, 170.95, -20) mm, rotated rx -180 ry 0 rz 0.01 deg; joints [33.817, -43.181, 99.032, -141.242, 62.786, 160.805] to (-250.31, 174.26, -20) mm, rotated rx 180 ry 0 rz 0.01 deg; joints [33.887, -43.038, 98.728, -141.117, 62.685, 160.657]
  MoveC 1418 to (-251.78, 177.57, -20) mm, rotated rx 180 ry 0 rz 0.01 deg; joints [33.958, -42.898, 98.429, -140.99, 62.586, 160.509] to (-254.77, 179.63, -20) mm, rotated rx -180 ry 0 rz 0.01 deg; joints [33.959, -42.73, 98.074, -140.928, 62.442, 160.376]
  MoveC 1419 to (-283.1, 193.5, -20) mm, rotated rx 180 ry 0 rz 0.01 deg; joints [33.804, -41.255, 94.969, -140.538, 61.122, 159.284] to (-307.01, 214.08, -20) mm, rotated rx -180 ry 0 rz 0.01 deg; joints [33.938, -39.732, 91.762, -139.786, 59.881, 157.973]
  MoveC 1420 to (-308.9, 214.54, -20) mm, rotated rx -180 ry 0 rz 0.01 deg; joints [33.914, -39.641, 91.572, -139.774, 59.796, 157.912] to (-310, 212.94, -20) mm, rotated rx -180 ry 0 rz 0.01 deg; joints [33.846, -39.639, 91.57, -139.846, 59.769, 157.949]
  MoveL 1421 to (-310, 144.51, -20) mm, rotated rx -180 ry 0 rz 0.01 deg; joints [31.794, -41.405, 95.361, -142.764, 60.577, 160.521]
  MoveC 1422 to (-308.9, 140.44, -20) mm, rotated rx -180 ry 0 rz 0.01 deg; joints [31.69, -41.549, 95.67, -142.931, 60.671, 160.691] to (-305.9, 137.47, -20) mm, rotated rx -180 ry 0 rz 0.01 deg; joints [31.655, -41.743, 96.08, -143.041, 60.831, 160.859]
  MoveC 1423 to (-294.92, 130.34, -20) mm, rotated rx 180 ry 0 rz 0.01 deg; joints [31.644, -42.358, 97.379, -143.279, 61.375, 161.333] to (-284.83, 121.97, -20) mm, rotated rx -180 ry 0 rz 0.01 deg; joints [31.576, -42.958, 98.65, -143.567, 61.891, 161.823]
  MoveC 1424 to (-275.67, 112.62, -20) mm, rotated rx 180 ry 0 rz 0.01 deg; joints [31.459, -43.537, 99.881, -143.897, 62.377, 162.319] to (-267.37, 102.5, -20) mm, rotated rx -180 ry 0 rz 0.01 deg; joints [31.298, -44.093, 101.066, -144.26, 62.835, 162.815]
  MoveC 1425 to (-264.01, 97.72, -20) mm, rotated rx 180 ry 0 rz 0.01 deg; joints [31.21, -44.331, 101.574, -144.434, 63.027, 163.036] to (-260.95, 92.76, -20) mm, rotated rx 180 ry 0 rz 0.01 deg; joints [31.109, -44.56, 102.066, -144.618, 63.209, 163.256]
  MoveL 1426 to (-246.6, 66.77, -20) mm, rotated rx 180 ry 0 rz 0.01 deg; joints [30.54, -45.676, 104.466, -145.588, 64.091, 164.351]
  MoveC 1427 to (-243.5, 63.66, -20) mm, rotated rx 180 ry 0 rz 0.01 deg; joints [30.498, -45.86, 104.86, -145.691, 64.252, 164.503] to (-239.25, 62.52, -20) mm, rotated rx -180 ry 0 rz 0.01 deg; joints [30.543, -46.044, 105.251, -145.699, 64.436, 164.611]
  MoveL 1428 to (-154.3, 62.52, -20) mm, rotated rx -180 ry 0 rz 0.01 deg; joints [32.295, -49.111, 111.769, -144.729, 67.755, 165.999]
  MoveC 1429 to (-150.05, 63.66, -20) mm, rotated rx -180 ry 0 rz 0.01 deg; joints [32.427, -49.235, 112.03, -144.625, 67.903, 166.032] to (-146.93, 66.77, -20) mm, rotated rx 180 ry 0 rz 0.01 deg; joints [32.601, -49.277, 112.114, -144.453, 67.983, 165.988]
  MoveL 1430 to (-132.32, 93.15, -20) mm, rotated rx -180 ry 0 rz 0.01 deg; joints [33.824, -49.211, 111.921, -143.153, 68.211, 165.42]
  MoveC 1431 to (-123.44, 106.36, -20) mm, rotated rx -180 ry 0 rz 0.01 deg; joints [34.471, -49.22, 111.915, -142.481, 68.378, 165.156] to (-112.88, 118.26, -20) mm, rotated rx -180 ry 0 rz 0.01 deg; joints [35.113, -49.308, 112.081, -141.837, 68.62, 164.958]
  MoveC 1432 to (-100.85, 128.68, -20) mm, rotated rx 180 ry 0 rz 0.01 deg; joints [35.743, -49.472, 112.411, -141.23, 68.929, 164.827] to (-87.61, 137.49, -20) mm, rotated rx 180 ry 0 rz 0.01 deg; joints [36.353, -49.705, 112.893, -140.664, 69.296, 164.766]
  MoveC 1433 to (-84.61, 140.48, -20) mm, rotated rx -180 ry 0 rz 0.01 deg; joints [36.524, -49.734, 112.948, -140.495, 69.366, 164.72] to (-83.52, 144.57, -20) mm, rotated rx 180 ry 0 rz 0.01 deg; joints [36.685, -49.674, 112.813, -140.312, 69.354, 164.608]
  MoveL 1434 to (-83.52, 212.94, -20) mm, rotated rx 180 ry 0 rz 0.01 deg; joints [38.864, -47.998, 109.119, -137.579, 68.501, 162.365]
  MoveC 1435 to (-84.62, 214.53, -20) mm, rotated rx 180 ry 0 rz 0.01 deg; joints [38.886, -47.921, 108.952, -137.533, 68.443, 162.292] to (-86.5, 214.08, -20) mm, rotated rx 180 ry 0 rz 0.01 deg; joints [38.825, -47.871, 108.847, -137.58, 68.382, 162.275]
  MoveC 1436 to (-101.26, 200.16, -20) mm, rotated rx -180 ry 0 rz 0.01 deg; joints [38.03, -47.736, 108.584, -138.355, 68.028, 162.493] to (-118.2, 189, -20) mm, rotated rx -180 ry 0 rz 0.01 deg; joints [37.273, -47.447, 107.991, -139.048, 67.555, 162.576]
  MoveC 1437 to (-136.7, 180.72, -20) mm, rotated rx -180 ry 0 rz 0.01 deg; joints [36.577, -47.02, 107.101, -139.635, 66.979, 162.533] to (-156.24, 175.34, -20) mm, rotated rx -180 ry 0 rz 0.01 deg; joints [35.957, -46.473, 105.954, -140.107, 66.319, 162.371]
  MoveC 1438 to (-170.81, 173.28, -20) mm, rotated rx 180 ry 0 rz 0.01 deg; joints [35.563, -46.009, 104.976, -140.368, 65.795, 162.181] to (-185.51, 172.77, -20) mm, rotated rx 180 ry 0 rz 0.01 deg; joints [35.221, -45.494, 103.891, -140.558, 65.242, 161.933]
  MoveL 1439 to (-214.9, 173.04, -20) mm, rotated rx 180 ry 0 rz 0.01 deg; joints [34.591, -44.411, 101.61, -140.854, 64.103, 161.381]
  MoveC 1440 to (-235.1, 174.69, -20) mm, rotated rx -180 ry 0 rz 0.01 deg; joints [34.216, -43.61, 99.925, -140.972, 63.287, 160.938] to (-254.77, 179.63, -20) mm, rotated rx -180 ry 0 rz 0.01 deg; joints [33.959, -42.73, 98.074, -140.928, 62.442, 160.376]
  MoveC 1441 to (-257.53, 181.62, -20) mm, rotated rx 180 ry 0 rz 0.01 deg; joints [33.963, -42.573, 97.741, -140.865, 62.307, 160.248] to (-258.69, 184.82, -20) mm, rotated rx 180 ry 0 rz 0.01 deg; joints [34.037, -42.446, 97.47, -140.74, 62.222, 160.109]
  MoveC 1442 to (-259.77, 188.02, -20) mm, rotated rx -180 ry 0 rz 0.01 deg; joints [34.111, -42.321, 97.204, -140.614, 62.14, 159.97] to (-262.38, 190.18, -20) mm, rotated rx 180 ry 0 rz 0.01 deg; joints [34.123, -42.164, 96.872, -140.543, 62.009, 159.838]
  MoveC 1443 to (-263.78, 190.81, -20) mm, rotated rx -180 ry 0 rz 0.01 deg; joints [34.114, -42.093, 96.721, -140.526, 61.944, 159.786] to (-265.17, 191.46, -20) mm, rotated rx -180 ry 0 rz 0.01 deg; joints [34.105, -42.021, 96.571, -140.509, 61.88, 159.734]
  MoveC 1444 to (-287.25, 205.04, -20) mm, rotated rx -180 ry 0 rz 0.01 deg; joints [34.064, -40.784, 93.968, -140.075, 60.813, 158.76] to (-305.91, 223.03, -20) mm, rotated rx 180 ry 0 rz 0.01 deg; joints [34.221, -39.533, 91.334, -139.399, 59.82, 157.648]
  MoveC 1445 to (-308.18, 225.95, -20) mm, rotated rx 180 ry 0 rz 0.01 deg; joints [34.261, -39.358, 90.966, -139.284, 59.69, 157.48] to (-310.25, 229.01, -20) mm, rotated rx 180 ry 0 rz 0.01 deg; joints [34.309, -39.187, 90.605, -139.161, 59.566, 157.311]
  MoveC 1446 to (-312.23, 232.12, -20) mm, rotated rx -180 ry 0 rz 0.01 deg; joints [34.36, -39.017, 90.247, -139.034, 59.444, 157.14] to (-314.27, 235.2, -20) mm, rotated rx -180 ry 0 rz 0.01 deg; joints [34.408, -38.845, 89.886, -138.909, 59.321, 156.968]
  MoveC 1447 to (-316, 235.82, -20) mm, rotated rx 180 ry 0 rz 0.01 deg; joints [34.392, -38.755, 89.696, -138.888, 59.24, 156.902] to (-317.1, 234.34, -20) mm, rotated rx 180 ry 0 rz 0.01 deg; joints [34.328, -38.75, 89.689, -138.955, 59.211, 156.935]
  MoveL 1448 to (-317.09, 140.15, -20) mm, rotated rx -180 ry 0 rz 0.01 deg; joints [31.526, -41.22, 94.983, -142.985, 60.327, 160.532]
  MoveC 1449 to (-315.96, 136.08, -20) mm, rotated rx 180 ry 0 rz 0.01 deg; joints [31.422, -41.366, 95.295, -143.154, 60.423, 160.703] to (-312.88, 133.18, -20) mm, rotated rx 180 ry 0 rz 0.01 deg; joints [31.391, -41.563, 95.71, -143.261, 60.587, 160.87]
  MoveC 1450 to (-292.13, 119.15, -20) mm, rotated rx -180 ry 0 rz 0.01 deg; joints [31.348, -42.735, 98.186, -143.736, 61.621, 161.779] to (-275.01, 100.86, -20) mm, rotated rx 180 ry 0 rz 0.01 deg; joints [31.097, -43.832, 100.521, -144.388, 62.54, 162.729]
  MoveC 1451 to (-272.92, 98.03, -20) mm, rotated rx 180 ry 0 rz 0.01 deg; joints [31.047, -43.978, 100.832, -144.492, 62.659, 162.863] to (-270.88, 95.16, -20) mm, rotated rx -180 ry 0 rz 0.01 deg; joints [30.994, -44.122, 101.14, -144.597, 62.775, 162.996]
  MoveC 1452 to (-268.93, 92.23, -20) mm, rotated rx -180 ry 0 rz 0.01 deg; joints [30.937, -44.264, 101.443, -144.706, 62.889, 163.129] to (-267.1, 89.22, -20) mm, rotated rx 180 ry 0 rz 0.01 deg; joints [30.875, -44.402, 101.739, -144.818, 62.999, 163.262]
  MoveL 1453 to (-250.69, 59.64, -20) mm, rotated rx 180 ry 0 rz 0.01 deg; joints [30.225, -45.673, 104.474, -145.926, 64.007, 164.508]
  MoveC 1454 to (-247.6, 56.55, -20) mm, rotated rx 180 ry 0 rz 0.01 deg; joints [30.182, -45.855, 104.864, -146.029, 64.168, 164.658] to (-243.39, 55.42, -20) mm, rotated rx 180 ry 0 rz 0.01 deg; joints [30.226, -46.038, 105.253, -146.037, 64.351, 164.765]
  MoveL 1455 to (-150.14, 55.42, -20) mm, rotated rx -180 ry 0 rz 0.01 deg; joints [32.141, -49.404, 112.408, -144.971, 67.998, 166.277]
  MoveC 1456 to (-145.94, 56.55, -20) mm, rotated rx 180 ry 0 rz 0.01 deg; joints [32.271, -49.525, 112.666, -144.867, 68.144, 166.309] to (-142.87, 59.62, -20) mm, rotated rx -180 ry 0 rz 0.01 deg; joints [32.444, -49.567, 112.749, -144.696, 68.223, 166.266]
  MoveL 1457 to (-126.17, 89.6, -20) mm, rotated rx 180 ry 0 rz 0.01 deg; joints [33.843, -49.497, 112.541, -143.213, 68.483, 165.628]
  MoveC 1458 to (-106.49, 114.66, -20) mm, rotated rx -180 ry 0 rz 0.01 deg; joints [35.143, -49.603, 112.718, -141.889, 68.898, 165.173] to (-80.6, 133.24, -20) mm, rotated rx -180 ry 0 rz 0.01 deg; joints [36.383, -50.033, 113.602, -140.724, 69.6, 165.013]
  MoveC 1459 to (-77.54, 136.1, -20) mm, rotated rx 180 ry 0 rz 0.01 deg; joints [36.552, -50.066, 113.668, -140.558, 69.673, 164.972] to (-76.42, 140.12, -20) mm, rotated rx -180 ry 0 rz 0.01 deg; joints [36.713, -50.009, 113.538, -140.377, 69.662, 164.864]
  MoveL 1460 to (-76.42, 234.34, -20) mm, rotated rx 180 ry 0 rz 0.01 deg; joints [39.699, -47.675, 108.397, -136.625, 68.485, 161.754]
  MoveC 1461 to (-77.52, 235.82, -20) mm, rotated rx 180 ry 0 rz 0.01 deg; joints [39.716, -47.6, 108.236, -136.584, 68.429, 161.684] to (-79.25, 235.2, -20) mm, rotated rx -180 ry 0 rz 0.01 deg; joints [39.654, -47.56, 108.152, -136.636, 68.375, 161.675]
  MoveC 1462 to (-84.84, 227.28, -20) mm, rotated rx 180 ry 0 rz 0.01 deg; joints [39.272, -47.584, 108.215, -137.033, 68.276, 161.851] to (-90.83, 219.67, -20) mm, rotated rx 180 ry 0 rz 0.01 deg; joints [38.89, -47.584, 108.228, -137.425, 68.159, 162.009]
  MoveC 1463 to (-97.42, 212.55, -20) mm, rotated rx -180 ry 0 rz 0.01 deg; joints [38.508, -47.549, 108.166, -137.806, 68.012, 162.138] to (-104.73, 206.18, -20) mm, rotated rx -180 ry 0 rz 0.01 deg; joints [38.132, -47.467, 108.005, -138.167, 67.829, 162.229]
  MoveC 1464 to (-118.75, 196.77, -20) mm, rotated rx 180 ry 0 rz 0.01 deg; joints [37.502, -47.233, 107.525, -138.744, 67.439, 162.304] to (-133.97, 189.44, -20) mm, rotated rx 180 ry 0 rz 0.01 deg; joints [36.914, -46.897, 106.826, -139.247, 66.973, 162.286]
  MoveC 1465 to (-150, 184.2, -20) mm, rotated rx 180 ry 0 rz 0.01 deg; joints [36.377, -46.472, 105.936, -139.669, 66.443, 162.181] to (-166.56, 180.94, -20) mm, rotated rx 180 ry 0 rz 0.01 deg; joints [35.898, -45.97, 104.882, -140.005, 65.863, 161.996]
  MoveC 1466 to (-172.57, 180.34, -20) mm, rotated rx -180 ry 0 rz 0.01 deg; joints [35.744, -45.771, 104.463, -140.101, 65.643, 161.909] to (-178.62, 180.13, -20) mm, rotated rx 180 ry 0 rz 0.01 deg; joints [35.603, -45.56, 104.018, -140.179, 65.416, 161.806]
  MoveL 1467 to (-214.9, 180.13, -20) mm, rotated rx -180 ry 0 rz 0.01 deg; joints [34.811, -44.234, 101.226, -140.562, 64.018, 161.133]
  MoveC 1468 to (-239.16, 182.67, -20) mm, rotated rx 180 ry 0 rz 0.01 deg; joints [34.375, -43.254, 99.167, -140.676, 63.031, 160.575] to (-262.38, 190.18, -20) mm, rotated rx -180 ry 0 rz 0.01 deg; joints [34.123, -42.164, 96.872, -140.543, 62.009, 159.838]
  MoveC 1469 to (-264.76, 192.25, -20) mm, rotated rx 180 ry 0 rz 0.01 deg; joints [34.137, -42.017, 96.56, -140.473, 61.887, 159.713] to (-265.58, 195.31, -20) mm, rotated rx 180 ry 0 rz 0.01 deg; joints [34.212, -41.905, 96.323, -140.35, 61.818, 159.584]
  MoveC 1470 to (-266.32, 198.36, -20) mm, rotated rx -180 ry 0 rz 0.01 deg; joints [34.289, -41.796, 96.09, -140.228, 61.751, 159.455] to (-268.56, 200.57, -20) mm, rotated rx 180 ry 0 rz 0.01 deg; joints [34.309, -41.65, 95.781, -140.15, 61.634, 159.326]
  MoveC 1471 to (-298.31, 224.41, -20) mm, rotated rx 180 ry 0 rz 0.01 deg; joints [34.412, -39.81, 91.907, -139.309, 60.122, 157.768] to (-318.26, 256.89, -20) mm, rotated rx 180 ry 0 rz 0.01 deg; joints [34.949, -38.056, 88.214, -137.987, 58.889, 155.987]
  MoveC 1472 to (-321.44, 258.63, -20) mm, rotated rx 180 ry 0 rz 0.01 deg; joints [34.936, -37.87, 87.825, -137.919, 58.732, 155.836] to (-323.74, 255.84, -20) mm, rotated rx -180 ry 0 rz 0.01 deg; joints [34.811, -37.852, 87.793, -138.045, 58.668, 155.894]
  MoveL 1473 to (-323.74, 135.89, -20) mm, rotated rx -180 ry 0 rz 0.01 deg; joints [31.27, -41.05, 94.635, -143.199, 60.094, 160.548]
  MoveC 1474 to (-322.64, 132, -20) mm, rotated rx -180 ry 0 rz 0.01 deg; joints [31.171, -41.189, 94.933, -143.361, 60.186, 160.712] to (-319.68, 129.25, -20) mm, rotated rx -180 ry 0 rz 0.01 deg; joints [31.142, -41.378, 95.331, -143.464, 60.344, 160.872]
  MoveL 1475 to (-311.69, 125.17, -20) mm, rotated rx -180 ry 0 rz 0.01 deg; joints [31.165, -41.803, 96.227, -143.597, 60.73, 161.18]
  MoveC 1476 to (-307.76, 122.99, -20) mm, rotated rx -180 ry 0 rz 0.01 deg; joints [31.171, -42.015, 96.673, -143.668, 60.921, 161.336] to (-304, 120.53, -20) mm, rotated rx 180 ry 0 rz 0.01 deg; joints [31.165, -42.225, 97.117, -143.751, 61.108, 161.498]
  MoveC 1477 to (-296.77, 114.82, -20) mm, rotated rx 180 ry 0 rz 0.01 deg; joints [31.124, -42.65, 98.017, -143.949, 61.477, 161.839] to (-290.16, 108.4, -20) mm, rotated rx -180 ry 0 rz 0.01 deg; joints [31.047, -43.063, 98.893, -144.178, 61.827, 162.188]
  MoveC 1478 to (-284.08, 101.49, -20) mm, rotated rx -180 ry 0 rz 0.01 deg; joints [30.943, -43.462, 99.742, -144.428, 62.159, 162.539] to (-278.37, 94.27, -20) mm, rotated rx -180 ry 0 rz 0.01 deg; joints [30.821, -43.85, 100.57, -144.692, 62.478, 162.888]
  MoveL 1479 to (-254.45, 52.84, -20) mm, rotated rx 180 ry 0 rz 0.01 deg; joints [29.926, -45.673, 104.487, -146.248, 63.932, 164.658]
  MoveC 1480 to (-251.56, 49.87, -20) mm, rotated rx 180 ry 0 rz 0.01 deg; joints [29.883, -45.845, 104.856, -146.347, 64.083, 164.801] to (-247.57, 48.78, -20) mm, rotated rx -180 ry 0 rz 0.01 deg; joints [29.923, -46.019, 105.226, -146.357, 64.258, 164.902]
  MoveL 1481 to (-145.93, 48.78, -20) mm, rotated rx 180 ry 0 rz 0.01 deg; joints [32.002, -49.686, 113.026, -145.192, 68.238, 166.539]
  MoveC 1482 to (-141.95, 49.87, -20) mm, rotated rx 180 ry 0 rz 0.01 deg; joints [32.127, -49.801, 113.269, -145.092, 68.375, 166.569] to (-139.09, 52.84, -20) mm, rotated rx 180 ry 0 rz 0.01 deg; joints [32.293, -49.838, 113.342, -144.927, 68.447, 166.526]
  MoveL 1483 to (-119.82, 86.74, -20) mm, rotated rx -180 ry 0 rz 0.01 deg; joints [33.891, -49.774, 113.138, -143.239, 68.753, 165.815]
  MoveC 1484 to (-108.5, 102.69, -20) mm, rotated rx 180 ry 0 rz 0.01 deg; joints [34.694, -49.804, 113.171, -142.411, 68.972, 165.51] to (-94.67, 116.53, -20) mm, rotated rx 180 ry 0 rz 0.01 deg; joints [35.486, -49.953, 113.464, -141.63, 69.304, 165.306]
  MoveC 1485 to (-89.82, 120.24, -20) mm, rotated rx -180 ry 0 rz 0.01 deg; joints [35.726, -50.029, 113.619, -141.401, 69.432, 165.269] to (-84.63, 123.47, -20) mm, rotated rx 180 ry 0 rz 0.01 deg; joints [35.959, -50.125, 113.819, -141.187, 69.578, 165.252]
  MoveC 1486 to (-79.28, 126.39, -20) mm, rotated rx 180 ry 0 rz 0.01 deg; joints [36.187, -50.233, 114.044, -140.981, 69.733, 165.247] to (-73.87, 129.22, -20) mm, rotated rx 180 ry 0 rz 0.01 deg; joints [36.414, -50.344, 114.276, -140.777, 69.89, 165.246]
  MoveC 1487 to (-70.88, 132, -20) mm, rotated rx -180 ry 0 rz 0.01 deg; joints [36.58, -50.376, 114.341, -140.614, 69.961, 165.207] to (-69.77, 135.93, -20) mm, rotated rx -180 ry 0 rz 0.01 deg; joints [36.738, -50.321, 114.215, -140.436, 69.95, 165.103]
  MoveL 1488 to (-69.78, 255.83, -20) mm, rotated rx 180 ry 0 rz 0.01 deg; joints [40.515, -47.319, 107.607, -135.682, 68.451, 161.12]
  MoveC 1489 to (-72.08, 258.62, -20) mm, rotated rx 180 ry 0 rz 0.01 deg; joints [40.539, -47.169, 107.285, -135.61, 68.336, 160.981] to (-75.25, 256.88, -20) mm, rotated rx 180 ry 0 rz 0.01 deg; joints [40.407, -47.112, 107.168, -135.726, 68.247, 160.986]
  MoveC 1490 to (-102.4, 217.04, -20) mm, rotated rx -180 ry 0 rz 0.01 deg; joints [38.525, -47.267, 107.562, -137.701, 67.779, 161.898] to (-143.84, 192.4, -20) mm, rotated rx 180 ry 0 rz 0.01 deg; joints [36.775, -46.482, 105.942, -139.258, 66.572, 162.011]
  MoveC 1491 to (-161.3, 188.19, -20) mm, rotated rx -180 ry 0 rz 0.01 deg; joints [36.243, -45.976, 104.88, -139.647, 65.973, 161.843] to (-179.21, 186.78, -20) mm, rotated rx -180 ry 0 rz 0.01 deg; joints [35.796, -45.373, 103.612, -139.915, 65.314, 161.566]
  MoveL 1492 to (-214.9, 186.78, -20) mm, rotated rx 180 ry 0 rz 0.01 deg; joints [35.015, -44.066, 100.863, -140.288, 63.938, 160.899]
  MoveC 1493 to (-242.6, 190.28, -20) mm, rotated rx 180 ry 0 rz 0.01 deg; joints [34.535, -42.929, 98.472, -140.388, 62.803, 160.234] to (-268.56, 200.57, -20) mm, rotated rx 180 ry 0 rz 0.01 deg; joints [34.309, -41.65, 95.781, -140.15, 61.634, 159.326]
  MoveC 1494 to (-271.66, 203.78, -20) mm, rotated rx -180 ry 0 rz 0.01 deg; joints [34.342, -41.443, 95.343, -140.035, 61.469, 159.141] to (-272.42, 208.18, -20) mm, rotated rx -180 ry 0 rz 0.01 deg; joints [34.457, -41.296, 95.031, -139.856, 61.386, 158.96]
  MoveC 1495 to (-273.03, 212.56, -20) mm, rotated rx -180 ry 0 rz 0.01 deg; joints [34.575, -41.156, 94.73, -139.676, 61.308, 158.782] to (-275.78, 216.02, -20) mm, rotated rx -180 ry 0 rz 0.01 deg; joints [34.621, -40.953, 94.302, -139.547, 61.154, 158.591]
  MoveC 1496 to (-297.22, 237.53, -20) mm, rotated rx -180 ry 0 rz 0.01 deg; joints [34.815, -39.491, 91.225, -138.746, 60.01, 157.276] to (-311.09, 264.55, -20) mm, rotated rx 180 ry 0 rz 0.01 deg; joints [35.309, -38.138, 88.372, -137.639, 59.1, 155.848]
  MoveC 1497 to (-313.2, 267.42, -20) mm, rotated rx -180 ry 0 rz 0.01 deg; joints [35.348, -37.964, 88.007, -137.521, 58.976, 155.676] to (-316.59, 268.52, -20) mm, rotated rx 180 ry 0 rz 0.01 deg; joints [35.311, -37.787, 87.638, -137.481, 58.818, 155.545]
  MoveL 1498 to (-329.25, 268.52, -20) mm, rotated rx 180 ry 0 rz 0.01 deg; joints [35.06, -37.241, 86.507, -137.504, 58.277, 155.222]
  MoveC 1499 to (-331.97, 267.39, -20) mm, rotated rx -180 ry 0 rz 0.01 deg; joints [34.975, -37.156, 86.333, -137.556, 58.173, 155.2] to (-333.1, 264.66, -20) mm, rotated rx 180 ry 0 rz 0.01 deg; joints [34.876, -37.187, 86.403, -137.676, 58.158, 155.286]
  MoveL 1500 to (-333.1, 129.76, -20) mm, rotated rx -180 ry 0 rz 0.01 deg; joints [30.909, -40.809, 94.142, -143.503, 59.764, 160.574]
  MoveC 1501 to (-331.97, 125.91, -20) mm, rotated rx 180 ry 0 rz 0.01 deg; joints [30.811, -40.949, 94.442, -143.664, 59.857, 160.738] to (-328.93, 123.27, -20) mm, rotated rx -180 ry 0 rz 0.01 deg; joints [30.786, -41.139, 94.842, -143.763, 60.018, 160.896]
  MoveC 1502 to (-319.51, 118.55, -20) mm, rotated rx 180 ry 0 rz 0.01 deg; joints [30.813, -41.64, 95.897, -143.92, 60.475, 161.257] to (-310.45, 113.16, -20) mm, rotated rx -180 ry 0 rz 0.01 deg; joints [30.814, -42.137, 96.945, -144.102, 60.921, 161.629]
  MoveC 1503 to (-302.01, 106.82, -20) mm, rotated rx -180 ry 0 rz 0.01 deg; joints [30.772, -42.626, 97.979, -144.322, 61.349, 162.015] to (-294.55, 99.34, -20) mm, rotated rx -180 ry 0 rz 0.01 deg; joints [30.676, -43.096, 98.977, -144.592, 61.748, 162.414]
  MoveC 1504 to (-284.36, 86.41, -20) mm, rotated rx -180 ry 0 rz 0.01 deg; joints [30.455, -43.79, 100.459, -145.069, 62.32, 163.041] to (-275.39, 72.6, -20) mm, rotated rx 180 ry 0 rz 0.01 deg; joints [30.178, -44.445, 101.861, -145.586, 62.849, 163.659]
  MoveC 1505 to (-267.42, 58.21, -20) mm, rotated rx -180 ry 0 rz 0.01 deg; joints [29.857, -45.063, 103.189, -146.132, 63.341, 164.265] to (-260.18, 43.44, -20) mm, rotated rx -180 ry 0 rz 0.01 deg; joints [29.504, -45.651, 104.457, -146.697, 63.805, 164.857]
  MoveC 1506 to (-257.63, 40.51, -20) mm, rotated rx 180 ry 0 rz 0.01 deg; joints [29.454, -45.809, 104.796, -146.799, 63.942, 164.992] to (-253.91, 39.42, -20) mm, rotated rx -180 ry 0 rz 0.01 deg; joints [29.488, -45.973, 105.145, -146.812, 64.107, 165.088]
  MoveL 1507 to (-139.56, 39.42, -20) mm, rotated rx 180 ry 0 rz 0.01 deg; joints [31.814, -50.096, 113.924, -145.498, 68.591, 166.911]
  MoveC 1508 to (-135.85, 40.51, -20) mm, rotated rx 180 ry 0 rz 0.01 deg; joints [31.933, -50.201, 114.146, -145.4, 68.718, 166.937] to (-133.32, 43.44, -20) mm, rotated rx 180 ry 0 rz 0.01 deg; joints [32.091, -50.227, 114.197, -145.241, 68.778, 166.89]
  MoveC 1509 to (-132.57, 45.1, -20) mm, rotated rx 180 ry 0 rz 0.01 deg; joints [32.166, -50.219, 114.176, -145.16, 68.786, 166.853] to (-131.83, 46.77, -20) mm, rotated rx 180 ry 0 rz 0.01 deg; joints [32.241, -50.21, 114.153, -145.08, 68.793, 166.816]
  MoveC 1510 to (-131.06, 48.43, -20) mm, rotated rx 180 ry 0 rz 0.01 deg; joints [32.316, -50.203, 114.134, -144.999, 68.802, 166.78] to (-130.19, 50.03, -20) mm, rotated rx 180 ry 0 rz 0.01 deg; joints [32.391, -50.199, 114.123, -144.919, 68.815, 166.746]
  MoveL 1511 to (-109.6, 85.22, -20) mm, rotated rx -180 ry 0 rz 0.01 deg; joints [34.075, -50.15, 113.946, -143.149, 69.148, 166.023]
  MoveC 1512 to (-97.22, 101.58, -20) mm, rotated rx -180 ry 0 rz 0.01 deg; joints [34.921, -50.203, 114.029, -142.283, 69.397, 165.724] to (-81.47, 114.72, -20) mm, rotated rx 180 ry 0 rz 0.01 deg; joints [35.743, -50.427, 114.482, -141.492, 69.801, 165.572]
  MoveC 1513 to (-77.41, 117.18, -20) mm, rotated rx 180 ry 0 rz 0.01 deg; joints [35.924, -50.503, 114.641, -141.325, 69.915, 165.561] to (-73.2, 119.34, -20) mm, rotated rx 180 ry 0 rz 0.01 deg; joints [36.1, -50.591, 114.825, -141.167, 70.038, 165.562]
  MoveC 1514 to (-68.9, 121.33, -20) mm, rotated rx -180 ry 0 rz 0.01 deg; joints [36.273, -50.684, 115.022, -141.014, 70.166, 165.569] to (-64.59, 123.29, -20) mm, rotated rx 180 ry 0 rz 0.01 deg; joints [36.445, -50.778, 115.221, -140.862, 70.294, 165.577]
  MoveC 1515 to (-61.55, 125.9, -20) mm, rotated rx -180 ry 0 rz 0.01 deg; joints [36.608, -50.816, 115.297, -140.704, 70.368, 165.545] to (-60.41, 129.75, -20) mm, rotated rx 180 ry 0 rz 0.01 deg; joints [36.765, -50.764, 115.178, -140.528, 70.359, 165.445]
  MoveL 1516 to (-60.42, 264.67, -20) mm, rotated rx -180 ry 0 rz 0.01 deg; joints [41.018, -47.382, 107.727, -135.19, 68.666, 160.971]
  MoveC 1517 to (-61.54, 267.4, -20) mm, rotated rx -180 ry 0 rz 0.01 deg; joints [41.07, -47.271, 107.488, -135.103, 68.593, 160.855] to (-64.27, 268.52, -20) mm, rotated rx -180 ry 0 rz 0.01 deg; joints [41.033, -47.153, 107.235, -135.103, 68.485, 160.767]
  MoveL 1518 to (-76.92, 268.52, -20) mm, rotated rx -180 ry 0 rz 0.01 deg; joints [40.71, -46.741, 106.363, -135.299, 68.044, 160.542]
  MoveC 1519 to (-80.31, 267.43, -20) mm, rotated rx -180 ry 0 rz 0.01 deg; joints [40.592, -46.66, 106.194, -135.393, 67.939, 160.521] to (-82.42, 264.55, -20) mm, rotated rx -180 ry 0 rz 0.01 deg; joints [40.454, -46.669, 106.218, -135.537, 67.901, 160.586]
  MoveC 1520 to (-92.36, 243.42, -20) mm, rotated rx 180 ry 0 rz 0.01 deg; joints [39.574, -46.91, 106.762, -136.512, 67.811, 161.158] to (-107.05, 225.27, -20) mm, rotated rx 180 ry 0 rz 0.01 deg; joints [38.663, -46.898, 106.766, -137.442, 67.511, 161.532]
  MoveC 1521 to (-125.53, 211.02, -20) mm, rotated rx -180 ry 0 rz 0.01 deg; joints [37.781, -46.64, 106.245, -138.267, 67.017, 161.697] to (-146.75, 201.3, -20) mm, rotated rx -180 ry 0 rz 0.01 deg; joints [36.983, -46.155, 105.238, -138.936, 66.356, 161.653]
  MoveC 1522 to (-163.47, 197.3, -20) mm, rotated rx 180 ry 0 rz 0.01 deg; joints [36.475, -45.669, 104.218, -139.304, 65.781, 161.489] to (-180.62, 196.03, -20) mm, rotated rx -180 ry 0 rz 0.01 deg; joints [36.049, -45.089, 102.997, -139.554, 65.148, 161.218]
  MoveL 1523 to (-214.9, 196.14, -20) mm, rotated rx -180 ry 0 rz 0.01 deg; joints [35.301, -43.828, 100.347, -139.903, 63.826, 160.566]
  MoveC 1524 to (-245.91, 200.91, -20) mm, rotated rx 180 ry 0 rz 0.01 deg; joints [34.787, -42.527, 97.613, -139.973, 62.544, 159.78] to (-274.06, 214.79, -20) mm, rotated rx 180 ry 0 rz 0.01 deg; joints [34.619, -41.055, 94.516, -139.588, 61.24, 158.675]
  MoveC 1525 to (-274.92, 215.4, -20) mm, rotated rx -180 ry 0 rz 0.01 deg; joints [34.62, -41.004, 94.409, -139.568, 61.197, 158.633] to (-275.78, 216.02, -20) mm, rotated rx 180 ry 0 rz 0.01 deg; joints [34.621, -40.953, 94.302, -139.547, 61.154, 158.591]
  MoveC 1526 to (-278.63, 219.89, -20) mm, rotated rx -180 ry 0 rz 0.01 deg; joints [34.677, -40.734, 93.839, -139.4, 60.991, 158.381] to (-278.78, 224.7, -20) mm, rotated rx -180 ry 0 rz 0.01 deg; joints [34.815, -40.598, 93.548, -139.199, 60.927, 158.193]
  MoveC 1527 to (-278.73, 229.45, -20) mm, rotated rx -180 ry 0 rz 0.01 deg; joints [34.955, -40.47, 93.273, -138.998, 60.872, 158.011] to (-281.09, 233.58, -20) mm, rotated rx 180 ry 0 rz 0.01 deg; joints [35.027, -40.261, 92.832, -138.837, 60.726, 157.798]
  MoveC 1528 to (-283.58, 236.18, -20) mm, rotated rx -180 ry 0 rz 0.01 deg; joints [35.052, -40.088, 92.468, -138.74, 60.592, 157.64] to (-285.97, 238.86, -20) mm, rotated rx 180 ry 0 rz 0.01 deg; joints [35.081, -39.916, 92.105, -138.639, 60.461, 157.481]
  MoveC 1529 to (-297.05, 255.28, -20) mm, rotated rx 180 ry 0 rz 0.01 deg; joints [35.328, -38.996, 90.167, -137.99, 59.803, 156.568] to (-303.97, 273.84, -20) mm, rotated rx 180 ry 0 rz 0.01 deg; joints [35.714, -38.165, 88.416, -137.22, 59.287, 155.638]
  MoveC 1530 to (-305.84, 276.75, -20) mm, rotated rx 180 ry 0 rz 0.01 deg; joints [35.758, -38, 88.068, -137.101, 59.173, 155.47] to (-309.12, 277.88, -20) mm, rotated rx -180 ry 0 rz 0.01 deg; joints [35.724, -37.827, 87.709, -137.06, 59.021, 155.341]
  MoveL 1531 to (-338.61, 277.88, -20) mm, rotated rx -180 ry 0 rz 0.01 deg; joints [35.138, -36.549, 85.061, -137.102, 57.757, 154.575]
  MoveC 1532 to (-341.34, 276.75, -20) mm, rotated rx -180 ry 0 rz 0.01 deg; joints [35.053, -36.463, 84.884, -137.153, 57.653, 154.551] to (-342.46, 274.03, -20) mm, rotated rx 180 ry 0 rz 0.01 deg; joints [34.955, -36.495, 84.956, -137.273, 57.637, 154.638]
  MoveL 1533 to (-342.46, 123.08, -20) mm, rotated rx 180 ry 0 rz 0.01 deg; joints [30.532, -40.577, 93.67, -143.827, 59.436, 160.62]
  MoveC 1534 to (-341.37, 119.55, -20) mm, rotated rx -180 ry 0 rz 0.01 deg; joints [30.443, -40.707, 93.948, -143.975, 59.524, 160.771] to (-338.48, 117.24, -20) mm, rotated rx 180 ry 0 rz 0.01 deg; joints [30.425, -40.884, 94.32, -144.063, 59.676, 160.914]
  MoveC 1535 to (-329.77, 113.47, -20) mm, rotated rx 180 ry 0 rz 0.01 deg; joints [30.466, -41.336, 95.271, -144.187, 60.094, 161.229] to (-321.34, 109.11, -20) mm, rotated rx 180 ry 0 rz 0.01 deg; joints [30.485, -41.787, 96.22, -144.333, 60.505, 161.554]
  MoveC 1536 to (-313.35, 103.95, -20) mm, rotated rx 180 ry 0 rz 0.01 deg; joints [30.471, -42.233, 97.162, -144.51, 60.904, 161.893] to (-306.06, 97.85, -20) mm, rotated rx 180 ry 0 rz 0.01 deg; joints [30.413, -42.668, 98.085, -144.728, 61.282, 162.245]
  MoveC 1537 to (-295.38, 86.02, -20) mm, rotated rx 180 ry 0 rz 0.01 deg; joints [30.235, -43.363, 99.562, -145.163, 61.865, 162.85] to (-286.67, 72.68, -20) mm, rotated rx 180 ry 0 rz 0.01 deg; joints [29.968, -44.002, 100.929, -145.668, 62.381, 163.454]
  MoveL 1538 to (-271.1, 44.98, -20) mm, rotated rx -180 ry 0 rz 0.01 deg; joints [29.35, -45.199, 103.501, -146.723, 63.339, 164.623]
  MoveC 1539 to (-269.73, 42.37, -20) mm, rotated rx 180 ry 0 rz 0.01 deg; joints [29.289, -45.306, 103.732, -146.823, 63.425, 164.729] to (-268.58, 39.66, -20) mm, rotated rx 180 ry 0 rz 0.01 deg; joints [29.22, -45.407, 103.948, -146.929, 63.503, 164.834]
  MoveC 1540 to (-267.54, 36.91, -20) mm, rotated rx 180 ry 0 rz 0.01 deg; joints [29.148, -45.503, 104.158, -147.037, 63.577, 164.938] to (-266.47, 34.17, -20) mm, rotated rx -180 ry 0 rz 0.01 deg; joints [29.076, -45.601, 104.369, -147.144, 63.652, 165.041]
  MoveC 1541 to (-264.08, 31.18, -20) mm, rotated rx -180 ry 0 rz 0.01 deg; joints [29.02, -45.753, 104.697, -147.251, 63.784, 165.174] to (-260.42, 30.05, -20) mm, rotated rx 180 ry 0 rz 0.01 deg; joints [29.051, -45.916, 105.043, -147.267, 63.947, 165.27]
  MoveL 1542 to (-133.1, 30.05, -20) mm, rotated rx -180 ry 0 rz 0.01 deg; joints [31.624, -50.505, 114.821, -145.802, 68.948, 167.28]
  MoveC 1543 to (-129.47, 31.16, -20) mm, rotated rx -180 ry 0 rz 0.01 deg; joints [31.743, -50.606, 115.037, -145.703, 69.071, 167.304] to (-127.07, 34.11, -20) mm, rotated rx -180 ry 0 rz 0.01 deg; joints [31.9, -50.628, 115.078, -145.544, 69.125, 167.256]
  MoveC 1544 to (-125.93, 36.97, -20) mm, rotated rx -180 ry 0 rz 0.01 deg; joints [32.027, -50.609, 115.031, -145.407, 69.133, 167.191] to (-124.84, 39.85, -20) mm, rotated rx 180 ry 0 rz 0.01 deg; joints [32.152, -50.588, 114.98, -145.27, 69.139, 167.124]
  MoveC 1545 to (-123.64, 42.69, -20) mm, rotated rx 180 ry 0 rz 0.01 deg; joints [32.279, -50.571, 114.936, -145.133, 69.149, 167.06] to (-122.21, 45.42, -20) mm, rotated rx 180 ry 0 rz 0.01 deg; joints [32.407, -50.563, 114.915, -144.997, 69.169, 167.003]
  MoveL 1546 to (-103.06, 78.56, -20) mm, rotated rx 180 ry 0 rz 0.01 deg; joints [33.997, -50.511, 114.734, -143.325, 69.47, 166.325]
  MoveC 1547 to (-91.35, 94.29, -20) mm, rotated rx 180 ry 0 rz 0.01 deg; joints [34.813, -50.557, 114.802, -142.49, 69.701, 166.037] to (-76.32, 106.9, -20) mm, rotated rx -180 ry 0 rz 0.01 deg; joints [35.603, -50.769, 115.233, -141.728, 70.083, 165.893]
  MoveC 1548 to (-71.24, 109.97, -20) mm, rotated rx 180 ry 0 rz 0.01 deg; joints [35.831, -50.865, 115.433, -141.518, 70.226, 165.88] to (-65.94, 112.63, -20) mm, rotated rx 180 ry 0 rz 0.01 deg; joints [36.052, -50.976, 115.666, -141.32, 70.38, 165.883]
  MoveC 1549 to (-60.51, 115, -20) mm, rotated rx 180 ry 0 rz 0.01 deg; joints [36.267, -51.096, 115.921, -141.13, 70.542, 165.896] to (-55.03, 117.25, -20) mm, rotated rx 180 ry 0 rz 0.01 deg; joints [36.479, -51.221, 116.184, -140.943, 70.707, 165.914]
  MoveC 1550 to (-52.14, 119.55, -20) mm, rotated rx 180 ry 0 rz 0.01 deg; joints [36.63, -51.26, 116.265, -140.798, 70.779, 165.889] to (-51.05, 123.09, -20) mm, rotated rx 180 ry 0 rz 0.01 deg; joints [36.777, -51.215, 116.16, -140.636, 70.772, 165.798]
  MoveL 1551 to (-51.05, 274.03, -20) mm, rotated rx 180 ry 0 rz 0.01 deg; joints [41.538, -47.426, 107.805, -134.678, 68.872, 160.802]
  MoveC 1552 to (-52.18, 276.76, -20) mm, rotated rx -180 ry 0 rz 0.01 deg; joints [41.589, -47.315, 107.565, -134.591, 68.799, 160.685] to (-54.91, 277.89, -20) mm, rotated rx -180 ry 0 rz 0.01 deg; joints [41.551, -47.197, 107.313, -134.592, 68.692, 160.597]
  MoveL 1553 to (-84.43, 277.89, -20) mm, rotated rx -180 ry 0 rz 0.01 deg; joints [40.795, -46.235, 105.281, -135.048, 67.666, 160.07]
  MoveC 1554 to (-87.69, 276.75, -20) mm, rotated rx -180 ry 0 rz 0.01 deg; joints [40.68, -46.159, 105.121, -135.14, 67.565, 160.052] to (-89.55, 273.84, -20) mm, rotated rx 180 ry 0 rz 0.01 deg; joints [40.548, -46.178, 105.166, -135.28, 67.535, 160.123]
  MoveC 1555 to (-97.53, 252.83, -20) mm, rotated rx -180 ry 0 rz 0.01 deg; joints [39.728, -46.486, 105.849, -136.218, 67.511, 160.733] to (-110.65, 234.58, -20) mm, rotated rx -180 ry 0 rz 0.01 deg; joints [38.858, -46.532, 105.977, -137.124, 67.266, 161.142]
  MoveC 1556 to (-127.95, 220.25, -20) mm, rotated rx -180 ry 0 rz 0.01 deg; joints [38.006, -46.319, 105.55, -137.931, 66.816, 161.334] to (-148.27, 210.66, -20) mm, rotated rx 180 ry 0 rz 0.01 deg; joints [37.235, -45.863, 104.605, -138.579, 66.186, 161.301]
  MoveC 1557 to (-155.69, 208.51, -20) mm, rotated rx -180 ry 0 rz 0.01 deg; joints [36.998, -45.658, 104.175, -138.757, 65.936, 161.241] to (-163.24, 206.88, -20) mm, rotated rx -180 ry 0 rz 0.01 deg; joints [36.775, -45.433, 103.704, -138.914, 65.673, 161.159]
